LIN {X 0,Y 206.682,Z 726.89,A -85,B 0,C 180,E1 -21277.278,E2 -21277.278} C_VEL
LIN {X 0,Y 209.321,Z 735.161,A -85,B 0,C 180,E1 -21281.538,E2 -21281.538} C_VEL
LIN {X 0,Y 210.247,Z 738.551,A -85,B 0,C 180,E1 -21283.14,E2 -21283.14} C_VEL
LIN {X 0,Y 210.147,Z 740.81,A -85,B 0,C 180,E1 -21284.029,E2 -21284.029} C_VEL
LIN {X 0,Y 208.364,Z 745.04,A -85,B 0,C 180,E1 -21285.371,E2 -21285.371} C_VEL
LIN {X 0,Y 206.552,Z 749.333,A -85,B 0,C 180,E1 -21286.732,E2 -21286.732} C_VEL
LIN {X 0,Y 206.448,Z 751.668,A -85,B 0,C 180,E1 -21287.635,E2 -21287.635} C_VEL
LIN {X 0,Y 206.909,Z 753.554,A -85,B 0,C 180,E1 -21288.438,E2 -21288.438} C_VEL
LIN {X 0,Y 209.343,Z 758.765,A -85,B 0,C 180,E1 -21289.235,E2 -21289.235} C_VEL
LIN {X 0,Y 216.039,Z 774.038,A -85,B 0,C 180,E1 -21291.329,E2 -21291.329} C_VEL
LIN {X 0,Y 217.099,Z 777.167,A -85,B 0,C 180,E1 -21291.673,E2 -21291.673} C_VEL
LIN {X 0,Y 219.836,Z 802.695,A -85,B 0,C 180,E1 -21293.228,E2 -21293.228} C_VEL
LIN {X 0,Y 222.118,Z 834.204,A -85,B 0,C 180,E1 -21294.866,E2 -21294.866} C_VEL
LIN {X 0,Y 222.467,Z 842.853,A -85,B 0,C 180,E1 -21295.257,E2 -21295.257} C_VEL
LIN {X 0,Y 221.203,Z 868.34,A -85,B 0,C 180,E1 -21296.1,E2 -21296.1} C_VEL
LIN {X 0,Y 219.69,Z 881.832,A -85,B 0,C 180,E1 -21296.868,E2 -21296.868} C_VEL
LIN {X 0,Y 217.809,Z 893.498,A -85,B 0,C 180,E1 -21297.849,E2 -21297.849} C_VEL
LIN {X 0,Y 215.482,Z 904.646,A -85,B 0,C 180,E1 -21299.107,E2 -21299.107} C_VEL
LIN {X 0,Y 212.493,Z 916.272,A -85,B 0,C 180,E1 -21300.818,E2 -21300.818} C_VEL
LIN {X 0,Y 209.467,Z 926.778,A -85,B 0,C 180,E1 -21302.814,E2 -21302.814} C_VEL
LIN {X 0,Y 206.798,Z 935.404,A -85,B 0,C 180,E1 -21304.877,E2 -21304.877} C_VEL
LIN {X 0,Y 204.268,Z 943.402,A -85,B 0,C 180,E1 -21307.244,E2 -21307.244} C_VEL
LIN {X 0,Y 201.734,Z 951.707,A -85,B 0,C 180,E1 -21310.359,E2 -21310.359} C_VEL
LIN {X 0,Y 199.924,Z 958.604,A -85,B 0,C 180,E1 -21313.682,E2 -21313.682} C_VEL
LIN {X 0,Y 198.895,Z 963.537,A -85,B 0,C 180,E1 -21316.737,E2 -21316.737} C_VEL
LIN {X 0,Y 198.461,Z 967.368,A -85,B 0,C 180,E1 -21319.816,E2 -21319.816} C_VEL
LIN {X 0,Y 198.565,Z 969.739,A -85,B 0,C 180,E1 -21322.322,E2 -21322.322} C_VEL
LIN {X 0,Y 199.067,Z 972.036,A -85,B 0,C 180,E1 -21325.965,E2 -21325.965} C_VEL
LIN {X 0,Y 199.324,Z 972.723,A -85,B 0,C 180,E1 -21327.993,E2 -21327.993} C_VEL
LIN {X 0,Y 199.612,Z 972.988,A -85,B 0,C 180,E1 -21330.013,E2 -21330.013} C_VEL
LIN {X 0,Y 199.315,Z 972.703,A -85,B 0,C 180,E1 -21332.034,E2 -21332.034} C_VEL
LIN {X 0,Y 199.032,Z 971.999,A -85,B 0,C 180,E1 -21334.063,E2 -21334.063} C_VEL
LIN {X 0,Y 198.567,Z 969.697,A -85,B 0,C 180,E1 -21337.684,E2 -21337.684} C_VEL
LIN {X 0,Y 198.778,Z 965.514,A -85,B 0,C 180,E1 -21341.743,E2 -21341.743} C_VEL
LIN {X 0,Y 198.912,Z 964.926,A -85,B 0,C 180,E1 -21342.252,E2 -21342.252} C_VEL
LIN {X 0,Y 199.993,Z 963.252,A -85,B 0,C 180,E1 -21346.34,E2 -21346.34} C_VEL
LIN {X 0,Y 200.983,Z 961.887,A -85,B 0,C 180,E1 -21348.356,E2 -21348.356} C_VEL
LIN {X 0,Y 204.209,Z 958.13,A -85,B 0,C 180,E1 -21352.258,E2 -21352.258} C_VEL
LIN {X 0,Y 207.427,Z 954.488,A -85,B 0,C 180,E1 -21355.069,E2 -21355.069} C_VEL
LIN {X 0,Y 212.837,Z 948.196,A -85,B 0,C 180,E1 -21358.619,E2 -21358.619} C_VEL
LIN {X 0,Y 217.816,Z 942.411,A -85,B 0,C 180,E1 -21361.093,E2 -21361.093} C_VEL
LIN {X 0,Y 223.39,Z 935.631,A -85,B 0,C 180,E1 -21363.417,E2 -21363.417} C_VEL
LIN {X 0,Y 229.603,Z 927.592,A -85,B 0,C 180,E1 -21365.573,E2 -21365.573} C_VEL
LIN {X 0,Y 235.263,Z 919.853,A -85,B 0,C 180,E1 -21367.235,E2 -21367.235} C_VEL
LIN {X 0,Y 241.992,Z 909.858,A -85,B 0,C 180,E1 -21368.916,E2 -21368.916} C_VEL
LIN {X 0,Y 247.802,Z 900.362,A -85,B 0,C 180,E1 -21370.193,E2 -21370.193} C_VEL
LIN {X 0,Y 253.695,Z 889.722,A -85,B 0,C 180,E1 -21371.324,E2 -21371.324} C_VEL
LIN {X 0,Y 259.007,Z 879.001,A -85,B 0,C 180,E1 -21372.199,E2 -21372.199} C_VEL
LIN {X 0,Y 264.829,Z 865.221,A -85,B 0,C 180,E1 -21373.116,E2 -21373.116} C_VEL
LIN {X 0,Y 269.77,Z 850.878,A -85,B 0,C 180,E1 -21373.951,E2 -21373.951} C_VEL
LIN {X 0,Y 272.98,Z 838.674,A -85,B 0,C 180,E1 -21374.9,E2 -21374.9} C_VEL
LIN {X 0,Y 276.113,Z 825.678,A -85,B 0,C 180,E1 -21376.168,E2 -21376.168} C_VEL
LIN {X 0,Y 277.691,Z 819.801,A -85,B 0,C 180,E1 -21376.838,E2 -21376.838} C_VEL
LIN {X 0,Y 277.681,Z 819.973,A -85,B 0,C 180,E1 -21377.153,E2 -21377.153} C_VEL
LIN {X 0,Y 272.848,Z 838.879,A -85,B 0,C 180,E1 -21378.34,E2 -21378.34} C_VEL
LIN {X 0,Y 269.797,Z 848.885,A -85,B 0,C 180,E1 -21379.119,E2 -21379.119} C_VEL
LIN {X 0,Y 265.86,Z 859.286,A -85,B 0,C 180,E1 -21380.13,E2 -21380.13} C_VEL
LIN {X 0,Y 261.413,Z 869.331,A -85,B 0,C 180,E1 -21381.313,E2 -21381.313} C_VEL
LIN {X 0,Y 255.951,Z 879.698,A -85,B 0,C 180,E1 -21382.837,E2 -21382.837} C_VEL
LIN {X 0,Y 250.488,Z 888.462,A -85,B 0,C 180,E1 -21384.468,E2 -21384.468} C_VEL
LIN {X 0,Y 244.479,Z 896.754,A -85,B 0,C 180,E1 -21386.401,E2 -21386.401} C_VEL
LIN {X 0,Y 239.584,Z 902.654,A -85,B 0,C 180,E1 -21388.129,E2 -21388.129} C_VEL
LIN {X 0,Y 235.845,Z 906.785,A -85,B 0,C 180,E1 -21389.563,E2 -21389.563} C_VEL
LIN {X 0,Y 230.515,Z 911.827,A -85,B 0,C 180,E1 -21391.799,E2 -21391.799} C_VEL
LIN {X 0,Y 225.539,Z 915.826,A -85,B 0,C 180,E1 -21394.135,E2 -21394.135} C_VEL
LIN {X 0,Y 222.426,Z 917.98,A -85,B 0,C 180,E1 -21395.747,E2 -21395.747} C_VEL
LIN {X 0,Y 216.721,Z 920.844,A -85,B 0,C 180,E1 -21399.101,E2 -21399.101} C_VEL
LIN {X 0,Y 214.157,Z 921.719,A -85,B 0,C 180,E1 -21400.842,E2 -21400.842} C_VEL
LIN {X 0,Y 209.572,Z 922.218,A -85,B 0,C 180,E1 -21404.438,E2 -21404.438} C_VEL
LIN {X 0,Y 207.565,Z 921.861,A -85,B 0,C 180,E1 -21406.29,E2 -21406.29} C_VEL
LIN {X 0,Y 205.827,Z 921.101,A -85,B 0,C 180,E1 -21408.178,E2 -21408.178} C_VEL
LIN {X 0,Y 204.377,Z 919.916,A -85,B 0,C 180,E1 -21410.1,E2 -21410.1} C_VEL
LIN {X 0,Y 202.622,Z 917.373,A -85,B 0,C 180,E1 -21413.027,E2 -21413.027} C_VEL
LIN {X 0,Y 201.189,Z 913.896,A -85,B 0,C 180,E1 -21415.994,E2 -21415.994} C_VEL
LIN {X 0,Y 200.193,Z 909.353,A -85,B 0,C 180,E1 -21418.994,E2 -21418.994} C_VEL
LIN {X 0,Y 199.633,Z 903.656,A -85,B 0,C 180,E1 -21422.018,E2 -21422.018} C_VEL
LIN {X 0,Y 199.473,Z 896.674,A -85,B 0,C 180,E1 -21425.053,E2 -21425.053} C_VEL
LIN {X 0,Y 199.828,Z 889.762,A -85,B 0,C 180,E1 -21427.579,E2 -21427.579} C_VEL
LIN {X 0,Y 200.16,Z 883.329,A -85,B 0,C 180,E1 -21429.601,E2 -21429.601} C_VEL
LIN {X 0,Y 200.784,Z 873.815,A -85,B 0,C 180,E1 -21432.123,E2 -21432.123} C_VEL
LIN {X 0,Y 201.441,Z 864.862,A -85,B 0,C 180,E1 -21434.136,E2 -21434.136} C_VEL
LIN {X 0,Y 202.101,Z 855.689,A -85,B 0,C 180,E1 -21435.894,E2 -21435.894} C_VEL
LIN {X 0,Y 202.743,Z 846.48,A -85,B 0,C 180,E1 -21437.397,E2 -21437.397} C_VEL
LIN {X 0,Y 203.492,Z 835.433,A -85,B 0,C 180,E1 -21438.892,E2 -21438.892} C_VEL
LIN {X 0,Y 204.086,Z 825.218,A -85,B 0,C 180,E1 -21440.012,E2 -21440.012} C_VEL
LIN {X 0,Y 204.601,Z 813.625,A -85,B 0,C 180,E1 -21441.01,E2 -21441.01} C_VEL
LIN {X 0,Y 205.158,Z 794.728,A -85,B 0,C 180,E1 -21442.202,E2 -21442.202} C_VEL
LIN {X 0,Y 206.609,Z 752.336,A -85,B 0,C 180,E1 -21444.663,E2 -21444.663} C_VEL
LIN {X 0,Y 199.974,Z 728.514,A -85,B 0,C 180,E1 -21446.385,E2 -21446.385} C_VEL
LIN {X 0,Y 199.791,Z 727.599,A -85,B 0,C 180,E1 -21446.517,E2 -21446.517} C_VEL
LIN {X 0,Y 199.694,Z 727.61,A -85,B 0,C 180,E1 -21452.346,E2 -21452.346} C_VEL
LIN {X 0,Y 199.645,Z 727.612,A -85,B 0,C 180,E1 -21456.759,E2 -21456.759} C_VEL
LIN {X 0,Y 199.622,Z 727.614,A -85,B 0,C 180,E1 -21459.325,E2 -21459.325} C_VEL
LIN {X 0,Y 199.592,Z 727.617,A -85,B 0,C 180,E1 -21462.3,E2 -21462.3} C_VEL
LIN {X 0,Y 199.615,Z 727.614,A -85,B 0,C 180,E1 -21467.447,E2 -21467.447} C_VEL
LIN {X 0,Y 200.663,Z 730.57,A -85,B 0,C 180,E1 -21467.936,E2 -21467.936} C_VEL
LIN {X 0,Y 202.629,Z 732.841,A -85,B 0,C 180,E1 -21468.561,E2 -21468.561} C_VEL
LIN {X 0,Y 204.932,Z 736.34,A -85,B 0,C 180,E1 -21469.309,E2 -21469.309} C_VEL
LIN {X 0,Y 212.578,Z 748.515,A -85,B 0,C 180,E1 -21471.644,E2 -21471.644} C_VEL
LIN {X 0,Y 220.401,Z 762.544,A -85,B 0,C 180,E1 -21473.858,E2 -21473.858} C_VEL
LIN {X 0,Y 225.212,Z 772.505,A -85,B 0,C 180,E1 -21475.165,E2 -21475.165} C_VEL
LIN {X 0,Y 224.036,Z 814.186,A -85,B 0,C 180,E1 -21476.613,E2 -21476.613} C_VEL
LIN {X 0,Y 223.198,Z 827.888,A -85,B 0,C 180,E1 -21477.481,E2 -21477.481} C_VEL
LIN {X 0,Y 221.705,Z 840.335,A -85,B 0,C 180,E1 -21478.599,E2 -21478.599} C_VEL
LIN {X 0,Y 219.835,Z 851.709,A -85,B 0,C 180,E1 -21479.985,E2 -21479.985} C_VEL
LIN {X 0,Y 217.391,Z 863.141,A -85,B 0,C 180,E1 -21481.771,E2 -21481.771} C_VEL
LIN {X 0,Y 214.936,Z 873.23,A -85,B 0,C 180,E1 -21483.793,E2 -21483.793} C_VEL
LIN {X 0,Y 212.46,Z 882.258,A -85,B 0,C 180,E1 -21486.083,E2 -21486.083} C_VEL
LIN {X 0,Y 209.598,Z 891.036,A -85,B 0,C 180,E1 -21488.86,E2 -21488.86} C_VEL
LIN {X 0,Y 206.932,Z 898.699,A -85,B 0,C 180,E1 -21491.983,E2 -21491.983} C_VEL
LIN {X 0,Y 205.007,Z 904.459,A -85,B 0,C 180,E1 -21495.089,E2 -21495.089} C_VEL
LIN {X 0,Y 203.947,Z 907.393,A -85,B 0,C 180,E1 -21497.044,E2 -21497.044} C_VEL
LIN {X 0,Y 202.294,Z 910.949,A -85,B 0,C 180,E1 -21499.984,E2 -21499.984} C_VEL
LIN {X 0,Y 201.542,Z 912.771,A -85,B 0,C 180,E1 -21501.969,E2 -21501.969} C_VEL
LIN {X 0,Y 200.837,Z 915.075,A -85,B 0,C 180,E1 -21505.974,E2 -21505.974} C_VEL
LIN {X 0,Y 200.446,Z 915.911,A -85,B 0,C 180,E1 -21509.987,E2 -21509.987} C_VEL
LIN {X 0,Y 200.829,Z 915.143,A -85,B 0,C 180,E1 -21514,E2 -21514} C_VEL
LIN {X 0,Y 201.516,Z 912.91,A -85,B 0,C 180,E1 -21518.005,E2 -21518.005} C_VEL
LIN {X 0,Y 202.756,Z 910.086,A -85,B 0,C 180,E1 -21520.976,E2 -21520.976} C_VEL
LIN {X 0,Y 204.386,Z 906.255,A -85,B 0,C 180,E1 -21523.914,E2 -21523.914} C_VEL
LIN {X 0,Y 206.303,Z 900.776,A -85,B 0,C 180,E1 -21527.134,E2 -21527.134} C_VEL
LIN {X 0,Y 208.71,Z 893.957,A -85,B 0,C 180,E1 -21530.176,E2 -21530.176} C_VEL
LIN {X 0,Y 211.425,Z 885.922,A -85,B 0,C 180,E1 -21532.975,E2 -21532.975} C_VEL
LIN {X 0,Y 213.852,Z 877.695,A -85,B 0,C 180,E1 -21535.276,E2 -21535.276} C_VEL
LIN {X 0,Y 216.494,Z 867.509,A -85,B 0,C 180,E1 -21537.539,E2 -21537.539} C_VEL
LIN {X 0,Y 218.937,Z 857.028,A -85,B 0,C 180,E1 -21539.362,E2 -21539.362} C_VEL
LIN {X 0,Y 221.06,Z 845.742,A -85,B 0,C 180,E1 -21540.91,E2 -21540.91} C_VEL
LIN {X 0,Y 222.821,Z 833.772,A -85,B 0,C 180,E1 -21542.141,E2 -21542.141} C_VEL
LIN {X 0,Y 223.808,Z 820.26,A -85,B 0,C 180,E1 -21543.191,E2 -21543.191} C_VEL
LIN {X 0,Y 224.359,Z 807.45,A -85,B 0,C 180,E1 -21543.801,E2 -21543.801} C_VEL
LIN {X 0,Y 225.36,Z 772.626,A -85,B 0,C 180,E1 -21544.956,E2 -21544.956} C_VEL
LIN {X 0,Y 218.541,Z 759.044,A -85,B 0,C 180,E1 -21546.814,E2 -21546.814} C_VEL
LIN {X 0,Y 211.371,Z 746.467,A -85,B 0,C 180,E1 -21548.88,E2 -21548.88} C_VEL
LIN {X 0,Y 204.548,Z 735.867,A -85,B 0,C 180,E1 -21550.983,E2 -21550.983} C_VEL
LIN {X 0,Y 202.076,Z 732.119,A -85,B 0,C 180,E1 -21551.794,E2 -21551.794} C_VEL
LIN {X 0,Y 200.231,Z 729.623,A -85,B 0,C 180,E1 -21552.405,E2 -21552.405} C_VEL
LIN {X 0,Y 199.679,Z 727.604,A -85,B 0,C 180,E1 -21552.669,E2 -21552.669} C_VEL
LIN {X 0,Y 199.649,Z 727.607,A -85,B 0,C 180,E1 -21557.642,E2 -21557.642} C_VEL
LIN {X 0,Y 199.659,Z 727.607,A -85,B 0,C 180,E1 -21560.725,E2 -21560.725} C_VEL
LIN {X 0,Y 199.585,Z 727.612,A -85,B 0,C 180,E1 -21565.708,E2 -21565.708} C_VEL
LIN {X 0,Y 199.646,Z 727.616,A -85,B 0,C 180,E1 -21568.127,E2 -21568.127} C_VEL
LIN {X 0,Y 199.633,Z 727.614,A -85,B 0,C 180,E1 -21572.764,E2 -21572.764} C_VEL
LIN {X 0,Y 199.659,Z 727.602,A -85,B 0,C 180,E1 -21577.219,E2 -21577.219} C_VEL
LIN {X 0,Y 199.74,Z 727.589,A -85,B 0,C 180,E1 -21581.753,E2 -21581.753} C_VEL
LIN {X 0,Y 199.773,Z 727.602,A -85,B 0,C 180,E1 -21585.744,E2 -21585.744} C_VEL
LIN {X 0,Y 199.992,Z 727.557,A -85,B 0,C 180,E1 -21589.88,E2 -21589.88} C_VEL
LIN {X 0,Y 199.971,Z 727.576,A -85,B 0,C 180,E1 -21593.948,E2 -21593.948} C_VEL
LIN {X 0,Y 200.286,Z 727.534,A -85,B 0,C 180,E1 -21597.989,E2 -21597.989} C_VEL
LIN {X 0,Y 200.422,Z 727.525,A -85,B 0,C 180,E1 -21600,E2 -21600} C_VEL
LIN {X 0,Y 200.286,Z 727.525,A -85,B 0,C 180,E1 -21602.011,E2 -21602.011} C_VEL
LIN {X 0,Y 200.04,Z 727.557,A -85,B 0,C 180,E1 -21608.079,E2 -21608.079} C_VEL
LIN {X 0,Y 199.825,Z 727.596,A -85,B 0,C 180,E1 -21612.182,E2 -21612.182} C_VEL
LIN {X 0,Y 199.742,Z 727.601,A -85,B 0,C 180,E1 -21616.349,E2 -21616.349} C_VEL
LIN {X 0,Y 199.633,Z 727.601,A -85,B 0,C 180,E1 -21620.613,E2 -21620.613} C_VEL
LIN {X 0,Y 199.615,Z 727.609,A -85,B 0,C 180,E1 -21624.992,E2 -21624.992} C_VEL
LIN {X 0,Y 199.613,Z 727.61,A -85,B 0,C 180,E1 -21629.532,E2 -21629.532} C_VEL
LIN {X 0,Y 199.608,Z 727.621,A -85,B 0,C 180,E1 -21632.358,E2 -21632.358} C_VEL
LIN {X 0,Y 199.642,Z 727.699,A -85,B 0,C 180,E1 -21635.699,E2 -21635.699} C_VEL
LIN {X 0,Y 202.208,Z 735.817,A -85,B 0,C 180,E1 -21640.15,E2 -21640.15} C_VEL
LIN {X 0,Y 204.255,Z 743.119,A -85,B 0,C 180,E1 -21643.756,E2 -21643.756} C_VEL
LIN {X 0,Y 206.448,Z 751.668,A -85,B 0,C 180,E1 -21647.635,E2 -21647.635} C_VEL
LIN {X 0,Y 207.307,Z 754.167,A -85,B 0,C 180,E1 -21648.409,E2 -21648.409} C_VEL
LIN {X 0,Y 209.079,Z 758.994,A -85,B 0,C 180,E1 -21649.184,E2 -21649.184} C_VEL
LIN {X 0,Y 210.72,Z 766.498,A -85,B 0,C 180,E1 -21649.857,E2 -21649.857} C_VEL
LIN {X 0,Y 211.768,Z 780.813,A -85,B 0,C 180,E1 -21650.718,E2 -21650.718} C_VEL
LIN {X 0,Y 214.104,Z 803.757,A -85,B 0,C 180,E1 -21652.158,E2 -21652.158} C_VEL
LIN {X 0,Y 216.27,Z 834.897,A -85,B 0,C 180,E1 -21653.836,E2 -21653.836} C_VEL
LIN {X 0,Y 216.602,Z 842.778,A -85,B 0,C 180,E1 -21654.21,E2 -21654.21} C_VEL
LIN {X 0,Y 215.429,Z 866.419,A -85,B 0,C 180,E1 -21655.004,E2 -21655.004} C_VEL
LIN {X 0,Y 213.934,Z 879.662,A -85,B 0,C 180,E1 -21655.748,E2 -21655.748} C_VEL
LIN {X 0,Y 211.831,Z 892.491,A -85,B 0,C 180,E1 -21656.827,E2 -21656.827} C_VEL
LIN {X 0,Y 209.431,Z 903.639,A -85,B 0,C 180,E1 -21658.111,E2 -21658.111} C_VEL
LIN {X 0,Y 206.327,Z 915.264,A -85,B 0,C 180,E1 -21659.857,E2 -21659.857} C_VEL
LIN {X 0,Y 203.093,Z 925.755,A -85,B 0,C 180,E1 -21661.886,E2 -21661.886} C_VEL
LIN {X 0,Y 200.36,Z 934.389,A -85,B 0,C 180,E1 -21664.011,E2 -21664.011} C_VEL
LIN {X 0,Y 197.687,Z 942.383,A -85,B 0,C 180,E1 -21666.441,E2 -21666.441} C_VEL
LIN {X 0,Y 195.345,Z 949.874,A -85,B 0,C 180,E1 -21669.295,E2 -21669.295} C_VEL
LIN {X 0,Y 193.539,Z 955.688,A -85,B 0,C 180,E1 -21672.037,E2 -21672.037} C_VEL
LIN {X 0,Y 192.209,Z 961.006,A -85,B 0,C 180,E1 -21675.185,E2 -21675.185} C_VEL
LIN {X 0,Y 191.533,Z 965.201,A -85,B 0,C 180,E1 -21678.372,E2 -21678.372} C_VEL
LIN {X 0,Y 191.505,Z 968.884,A -85,B 0,C 180,E1 -21682.252,E2 -21682.252} C_VEL
LIN {X 0,Y 191.969,Z 971.021,A -85,B 0,C 180,E1 -21685.815,E2 -21685.815} C_VEL
LIN {X 0,Y 192.264,Z 971.716,A -85,B 0,C 180,E1 -21687.919,E2 -21687.919} C_VEL
LIN {X 0,Y 192.569,Z 971.983,A -85,B 0,C 180,E1 -21690.014,E2 -21690.014} C_VEL
LIN {X 0,Y 192.252,Z 971.695,A -85,B 0,C 180,E1 -21692.109,E2 -21692.109} C_VEL
LIN {X 0,Y 191.935,Z 970.984,A -85,B 0,C 180,E1 -21694.213,E2 -21694.213} C_VEL
LIN {X 0,Y 191.506,Z 968.843,A -85,B 0,C 180,E1 -21697.751,E2 -21697.751} C_VEL
LIN {X 0,Y 191.685,Z 965.136,A -85,B 0,C 180,E1 -21701.647,E2 -21701.647} C_VEL
LIN {X 0,Y 192.033,Z 963.462,A -85,B 0,C 180,E1 -21703.101,E2 -21703.101} C_VEL
LIN {X 0,Y 193.163,Z 962.18,A -85,B 0,C 180,E1 -21706.935,E2 -21706.935} C_VEL
LIN {X 0,Y 195.475,Z 959.665,A -85,B 0,C 180,E1 -21710.806,E2 -21710.806} C_VEL
LIN {X 0,Y 198.681,Z 956.637,A -85,B 0,C 180,E1 -21714.016,E2 -21714.016} C_VEL
LIN {X 0,Y 203.688,Z 951.595,A -85,B 0,C 180,E1 -21717.775,E2 -21717.775} C_VEL
LIN {X 0,Y 208.299,Z 946.892,A -85,B 0,C 180,E1 -21720.417,E2 -21720.417} C_VEL
LIN {X 0,Y 214.636,Z 940.191,A -85,B 0,C 180,E1 -21723.274,E2 -21723.274} C_VEL
LIN {X 0,Y 220.663,Z 933.395,A -85,B 0,C 180,E1 -21725.551,E2 -21725.551} C_VEL
LIN {X 0,Y 227.402,Z 925.323,A -85,B 0,C 180,E1 -21727.629,E2 -21727.629} C_VEL
LIN {X 0,Y 233.442,Z 917.617,A -85,B 0,C 180,E1 -21729.226,E2 -21729.226} C_VEL
LIN {X 0,Y 241.229,Z 906.64,A -85,B 0,C 180,E1 -21730.97,E2 -21730.97} C_VEL
LIN {X 0,Y 247.616,Z 896.668,A -85,B 0,C 180,E1 -21732.201,E2 -21732.201} C_VEL
LIN {X 0,Y 253.928,Z 885.682,A -85,B 0,C 180,E1 -21733.247,E2 -21733.247} C_VEL
LIN {X 0,Y 260.715,Z 872.156,A -85,B 0,C 180,E1 -21734.237,E2 -21734.237} C_VEL
LIN {X 0,Y 267.115,Z 856.327,A -85,B 0,C 180,E1 -21735.143,E2 -21735.143} C_VEL
LIN {X 0,Y 270.759,Z 845.161,A -85,B 0,C 180,E1 -21735.939,E2 -21735.939} C_VEL
LIN {X 0,Y 273.052,Z 837.373,A -85,B 0,C 180,E1 -21736.659,E2 -21736.659} C_VEL
LIN {X 0,Y 269.389,Z 849.095,A -85,B 0,C 180,E1 -21737.542,E2 -21737.542} C_VEL
LIN {X 0,Y 265.234,Z 859.664,A -85,B 0,C 180,E1 -21738.514,E2 -21738.514} C_VEL
LIN {X 0,Y 260.52,Z 869.771,A -85,B 0,C 180,E1 -21739.651,E2 -21739.651} C_VEL
LIN {X 0,Y 254.762,Z 880.196,A -85,B 0,C 180,E1 -21741.127,E2 -21741.127} C_VEL
LIN {X 0,Y 247.996,Z 890.406,A -85,B 0,C 180,E1 -21742.972,E2 -21742.972} C_VEL
LIN {X 0,Y 242.57,Z 897.51,A -85,B 0,C 180,E1 -21744.587,E2 -21744.587} C_VEL
LIN {X 0,Y 236.333,Z 904.531,A -85,B 0,C 180,E1 -21746.623,E2 -21746.623} C_VEL
LIN {X 0,Y 230.379,Z 910.327,A -85,B 0,C 180,E1 -21748.761,E2 -21748.761} C_VEL
LIN {X 0,Y 224.814,Z 914.954,A -85,B 0,C 180,E1 -21751.017,E2 -21751.017} C_VEL
LIN {X 0,Y 219.592,Z 918.523,A -85,B 0,C 180,E1 -21753.38,E2 -21753.38} C_VEL
LIN {X 0,Y 213.254,Z 921.885,A -85,B 0,C 180,E1 -21756.705,E2 -21756.705} C_VEL
LIN {X 0,Y 207.682,Z 923.485,A -85,B 0,C 180,E1 -21760.22,E2 -21760.22} C_VEL
LIN {X 0,Y 202.88,Z 923.594,A -85,B 0,C 180,E1 -21763.911,E2 -21763.911} C_VEL
LIN {X 0,Y 200.786,Z 923.028,A -85,B 0,C 180,E1 -21765.817,E2 -21765.817} C_VEL
LIN {X 0,Y 198.948,Z 922.046,A -85,B 0,C 180,E1 -21767.763,E2 -21767.763} C_VEL
LIN {X 0,Y 196.143,Z 918.897,A -85,B 0,C 180,E1 -21771.76,E2 -21771.76} C_VEL
LIN {X 0,Y 194.579,Z 915.419,A -85,B 0,C 180,E1 -21774.819,E2 -21774.819} C_VEL
LIN {X 0,Y 193.406,Z 910.946,A -85,B 0,C 180,E1 -21777.918,E2 -21777.918} C_VEL
LIN {X 0,Y 192.612,Z 904.231,A -85,B 0,C 180,E1 -21781.568,E2 -21781.568} C_VEL
LIN {X 0,Y 192.401,Z 897.087,A -85,B 0,C 180,E1 -21784.714,E2 -21784.714} C_VEL
LIN {X 0,Y 192.696,Z 890.026,A -85,B 0,C 180,E1 -21787.334,E2 -21787.334} C_VEL
LIN {X 0,Y 193.082,Z 883.516,A -85,B 0,C 180,E1 -21789.427,E2 -21789.427} C_VEL
LIN {X 0,Y 193.602,Z 874.958,A -85,B 0,C 180,E1 -21791.782,E2 -21791.782} C_VEL
LIN {X 0,Y 194.25,Z 865.987,A -85,B 0,C 180,E1 -21793.869,E2 -21793.869} C_VEL
LIN {X 0,Y 194.949,Z 856.821,A -85,B 0,C 180,E1 -21795.687,E2 -21795.687} C_VEL
LIN {X 0,Y 195.536,Z 847.567,A -85,B 0,C 180,E1 -21797.249,E2 -21797.249} C_VEL
LIN {X 0,Y 196.343,Z 836.551,A -85,B 0,C 180,E1 -21798.793,E2 -21798.793} C_VEL
LIN {X 0,Y 197.016,Z 825.184,A -85,B 0,C 180,E1 -21800.081,E2 -21800.081} C_VEL
LIN {X 0,Y 197.525,Z 813.614,A -85,B 0,C 180,E1 -21801.105,E2 -21801.105} C_VEL
LIN {X 0,Y 198.374,Z 783.132,A -85,B 0,C 180,E1 -21803.074,E2 -21803.074} C_VEL
LIN {X 0,Y 199.568,Z 753.543,A -85,B 0,C 180,E1 -21804.862,E2 -21804.862} C_VEL
LIN {X 0,Y 192.738,Z 728.477,A -85,B 0,C 180,E1 -21806.755,E2 -21806.755} C_VEL
LIN {X 0,Y 192.634,Z 728.487,A -85,B 0,C 180,E1 -21812.933,E2 -21812.933} C_VEL
LIN {X 0,Y 192.61,Z 728.488,A -85,B 0,C 180,E1 -21816.59,E2 -21816.59} C_VEL
LIN {X 0,Y 192.531,Z 728.496,A -85,B 0,C 180,E1 -21821.076,E2 -21821.076} C_VEL
LIN {X 0,Y 192.546,Z 728.505,A -85,B 0,C 180,E1 -21825.525,E2 -21825.525} C_VEL
LIN {X 0,Y 193.445,Z 731.172,A -85,B 0,C 180,E1 -21825.933,E2 -21825.933} C_VEL
LIN {X 0,Y 195.706,Z 733.846,A -85,B 0,C 180,E1 -21826.727,E2 -21826.727} C_VEL
LIN {X 0,Y 197.951,Z 737.299,A -85,B 0,C 180,E1 -21827.528,E2 -21827.528} C_VEL
LIN {X 0,Y 203.703,Z 745.873,A -85,B 0,C 180,E1 -21829.441,E2 -21829.441} C_VEL
LIN {X 0,Y 210.994,Z 758.159,A -85,B 0,C 180,E1 -21831.707,E2 -21831.707} C_VEL
LIN {X 0,Y 218.095,Z 771.897,A -85,B 0,C 180,E1 -21833.777,E2 -21833.777} C_VEL
LIN {X 0,Y 219.476,Z 774.961,A -85,B 0,C 180,E1 -21834.174,E2 -21834.174} C_VEL
LIN {X 0,Y 218.571,Z 805.347,A -85,B 0,C 180,E1 -21835.211,E2 -21835.211} C_VEL
LIN {X 0,Y 218.023,Z 819.467,A -85,B 0,C 180,E1 -21835.831,E2 -21835.831} C_VEL
LIN {X 0,Y 216.99,Z 831.806,A -85,B 0,C 180,E1 -21836.718,E2 -21836.718} C_VEL
LIN {X 0,Y 215.229,Z 844.578,A -85,B 0,C 180,E1 -21837.996,E2 -21837.996} C_VEL
LIN {X 0,Y 213.099,Z 856.132,A -85,B 0,C 180,E1 -21839.538,E2 -21839.538} C_VEL
LIN {X 0,Y 210.666,Z 866.582,A -85,B 0,C 180,E1 -21841.331,E2 -21841.331} C_VEL
LIN {X 0,Y 208.083,Z 876.168,A -85,B 0,C 180,E1 -21843.403,E2 -21843.403} C_VEL
LIN {X 0,Y 205.553,Z 884.854,A -85,B 0,C 180,E1 -21845.765,E2 -21845.765} C_VEL
LIN {X 0,Y 202.619,Z 893.348,A -85,B 0,C 180,E1 -21848.629,E2 -21848.629} C_VEL
LIN {X 0,Y 200.081,Z 900.104,A -85,B 0,C 180,E1 -21851.558,E2 -21851.558} C_VEL
LIN {X 0,Y 198.224,Z 905.463,A -85,B 0,C 180,E1 -21854.566,E2 -21854.566} C_VEL
LIN {X 0,Y 197.104,Z 908.397,A -85,B 0,C 180,E1 -21856.586,E2 -21856.586} C_VEL
LIN {X 0,Y 195.377,Z 911.953,A -85,B 0,C 180,E1 -21859.625,E2 -21859.625} C_VEL
LIN {X 0,Y 194.585,Z 913.774,A -85,B 0,C 180,E1 -21861.68,E2 -21861.68} C_VEL
LIN {X 0,Y 193.827,Z 916.078,A -85,B 0,C 180,E1 -21865.828,E2 -21865.828} C_VEL
LIN {X 0,Y 193.418,Z 916.914,A -85,B 0,C 180,E1 -21869.986,E2 -21869.986} C_VEL
LIN {X 0,Y 193.819,Z 916.145,A -85,B 0,C 180,E1 -21874.145,E2 -21874.145} C_VEL
LIN {X 0,Y 194.558,Z 913.912,A -85,B 0,C 180,E1 -21878.293,E2 -21878.293} C_VEL
LIN {X 0,Y 195.861,Z 911.088,A -85,B 0,C 180,E1 -21881.368,E2 -21881.368} C_VEL
LIN {X 0,Y 197.571,Z 907.256,A -85,B 0,C 180,E1 -21884.404,E2 -21884.404} C_VEL
LIN {X 0,Y 199.597,Z 901.777,A -85,B 0,C 180,E1 -21887.728,E2 -21887.728} C_VEL
LIN {X 0,Y 202.127,Z 894.958,A -85,B 0,C 180,E1 -21890.863,E2 -21890.863} C_VEL
LIN {X 0,Y 204.972,Z 886.922,A -85,B 0,C 180,E1 -21893.742,E2 -21893.742} C_VEL
LIN {X 0,Y 207.518,Z 878.694,A -85,B 0,C 180,E1 -21896.105,E2 -21896.105} C_VEL
LIN {X 0,Y 210.287,Z 868.507,A -85,B 0,C 180,E1 -21898.424,E2 -21898.424} C_VEL
LIN {X 0,Y 212.84,Z 858.026,A -85,B 0,C 180,E1 -21900.29,E2 -21900.29} C_VEL
LIN {X 0,Y 215.062,Z 846.738,A -85,B 0,C 180,E1 -21901.872,E2 -21901.872} C_VEL
LIN {X 0,Y 216.904,Z 834.766,A -85,B 0,C 180,E1 -21903.128,E2 -21903.128} C_VEL
LIN {X 0,Y 217.966,Z 821.212,A -85,B 0,C 180,E1 -21904.204,E2 -21904.204} C_VEL
LIN {X 0,Y 218.551,Z 808.547,A -85,B 0,C 180,E1 -21904.822,E2 -21904.822} C_VEL
LIN {X 0,Y 219.51,Z 774.785,A -85,B 0,C 180,E1 -21905.984,E2 -21905.984} C_VEL
LIN {X 0,Y 212.755,Z 761.39,A -85,B 0,C 180,E1 -21907.932,E2 -21907.932} C_VEL
LIN {X 0,Y 205.359,Z 748.49,A -85,B 0,C 180,E1 -21910.203,E2 -21910.203} C_VEL
LIN {X 0,Y 198.123,Z 737.387,A -85,B 0,C 180,E1 -21912.602,E2 -21912.602} C_VEL
LIN {X 0,Y 195.872,Z 734.06,A -85,B 0,C 180,E1 -21913.399,E2 -21913.399} C_VEL
LIN {X 0,Y 195.162,Z 733.067,A -85,B 0,C 180,E1 -21913.654,E2 -21913.654} C_VEL
LIN {X 0,Y 193.321,Z 730.758,A -85,B 0,C 180,E1 -21914.314,E2 -21914.314} C_VEL
LIN {X 0,Y 192.621,Z 728.459,A -85,B 0,C 180,E1 -21914.692,E2 -21914.692} C_VEL
LIN {X 0,Y 192.572,Z 728.495,A -85,B 0,C 180,E1 -21920.006,E2 -21920.006} C_VEL
LIN {X 0,Y 192.556,Z 728.497,A -85,B 0,C 180,E1 -21924.269,E2 -21924.269} C_VEL
LIN {X 0,Y 192.549,Z 728.495,A -85,B 0,C 180,E1 -21929.27,E2 -21929.27} C_VEL
LIN {X 0,Y 192.609,Z 728.479,A -85,B 0,C 180,E1 -21931.683,E2 -21931.683} C_VEL
LIN {X 0,Y 192.631,Z 728.475,A -85,B 0,C 180,E1 -21936.339,E2 -21936.339} C_VEL
LIN {X 0,Y 192.676,Z 728.471,A -85,B 0,C 180,E1 -21941.453,E2 -21941.453} C_VEL
LIN {X 0,Y 192.702,Z 728.481,A -85,B 0,C 180,E1 -21945.209,E2 -21945.209} C_VEL
LIN {X 0,Y 192.895,Z 728.439,A -85,B 0,C 180,E1 -21949.551,E2 -21949.551} C_VEL
LIN {X 0,Y 192.99,Z 728.445,A -85,B 0,C 180,E1 -21951.624,E2 -21951.624} C_VEL
LIN {X 0,Y 193.225,Z 728.412,A -85,B 0,C 180,E1 -21957.915,E2 -21957.915} C_VEL
LIN {X 0,Y 193.387,Z 728.401,A -85,B 0,C 180,E1 -21960,E2 -21960} C_VEL
LIN {X 0,Y 192.93,Z 728.445,A -85,B 0,C 180,E1 -21964.178,E2 -21964.178} C_VEL
LIN {X 0,Y 192.99,Z 728.433,A -85,B 0,C 180,E1 -21968.376,E2 -21968.376} C_VEL
LIN {X 0,Y 192.748,Z 728.478,A -85,B 0,C 180,E1 -21972.637,E2 -21972.637} C_VEL
LIN {X 0,Y 192.697,Z 728.478,A -85,B 0,C 180,E1 -21976.964,E2 -21976.964} C_VEL
LIN {X 0,Y 192.57,Z 728.481,A -85,B 0,C 180,E1 -21981.405,E2 -21981.405} C_VEL
LIN {X 0,Y 192.602,Z 728.49,A -85,B 0,C 180,E1 -21984.225,E2 -21984.225} C_VEL
LIN {X 0,Y 192.593,Z 728.49,A -85,B 0,C 180,E1 -21988.897,E2 -21988.897} C_VEL
LIN {X 0,Y 192.54,Z 728.587,A -85,B 0,C 180,E1 -21993.982,E2 -21993.982} C_VEL
LIN {X 0,Y 194.97,Z 736.132,A -85,B 0,C 180,E1 -21998.448,E2 -21998.448} C_VEL
LIN {X 0,Y 197.279,Z 743.979,A -85,B 0,C 180,E1 -22002.599,E2 -22002.599} C_VEL
LIN {X 0,Y 199.32,Z 752.073,A -85,B 0,C 180,E1 -22006.472,E2 -22006.472} C_VEL
LIN {X 0,Y 201.999,Z 757.443,A -85,B 0,C 180,E1 -22007.416,E2 -22007.416} C_VEL
LIN {X 0,Y 207.74,Z 770.058,A -85,B 0,C 180,E1 -22009.364,E2 -22009.364} C_VEL
LIN {X 0,Y 211.641,Z 779.541,A -85,B 0,C 180,E1 -22010.637,E2 -22010.637} C_VEL
LIN {X 0,Y 211.768,Z 780.813,A -85,B 0,C 180,E1 -22010.718,E2 -22010.718} C_VEL
LIN {X 0,Y 211.798,Z 786.652,A -85,B 0,C 180,E1 -22010.971,E2 -22010.971} C_VEL
LIN {X 0,Y 209.112,Z 806.31,A -85,B 0,C 180,E1 -22011.235,E2 -22011.235} C_VEL
LIN {X 0,Y 209.019,Z 812.183,A -85,B 0,C 180,E1 -22011.464,E2 -22011.464} C_VEL
LIN {X 0,Y 210.826,Z 842.002,A -85,B 0,C 180,E1 -22013.08,E2 -22013.08} C_VEL
LIN {X 0,Y 209.552,Z 866.277,A -85,B 0,C 180,E1 -22013.927,E2 -22013.927} C_VEL
LIN {X 0,Y 207.957,Z 879.673,A -85,B 0,C 180,E1 -22014.717,E2 -22014.717} C_VEL
LIN {X 0,Y 205.859,Z 891.474,A -85,B 0,C 180,E1 -22015.733,E2 -22015.733} C_VEL
LIN {X 0,Y 203.441,Z 902.632,A -85,B 0,C 180,E1 -22017.055,E2 -22017.055} C_VEL
LIN {X 0,Y 200.22,Z 914.255,A -85,B 0,C 180,E1 -22018.837,E2 -22018.837} C_VEL
LIN {X 0,Y 196.851,Z 924.744,A -85,B 0,C 180,E1 -22020.911,E2 -22020.911} C_VEL
LIN {X 0,Y 193.982,Z 933.376,A -85,B 0,C 180,E1 -22023.089,E2 -22023.089} C_VEL
LIN {X 0,Y 191.146,Z 941.364,A -85,B 0,C 180,E1 -22025.584,E2 -22025.584} C_VEL
LIN {X 0,Y 188.43,Z 949.498,A -85,B 0,C 180,E1 -22028.819,E2 -22028.819} C_VEL
LIN {X 0,Y 186.187,Z 956.559,A -85,B 0,C 180,E1 -22032.44,E2 -22032.44} C_VEL
LIN {X 0,Y 184.954,Z 961.492,A -85,B 0,C 180,E1 -22035.716,E2 -22035.716} C_VEL
LIN {X 0,Y 184.403,Z 965.329,A -85,B 0,C 180,E1 -22039.03,E2 -22039.03} C_VEL
LIN {X 0,Y 184.456,Z 968.012,A -85,B 0,C 180,E1 -22042.153,E2 -22042.153} C_VEL
LIN {X 0,Y 184.875,Z 970.007,A -85,B 0,C 180,E1 -22045.654,E2 -22045.654} C_VEL
LIN {X 0,Y 185.199,Z 970.707,A -85,B 0,C 180,E1 -22047.84,E2 -22047.84} C_VEL
LIN {X 0,Y 185.524,Z 970.978,A -85,B 0,C 180,E1 -22050.014,E2 -22050.014} C_VEL
LIN {X 0,Y 185.184,Z 970.686,A -85,B 0,C 180,E1 -22052.189,E2 -22052.189} C_VEL
LIN {X 0,Y 184.842,Z 969.968,A -85,B 0,C 180,E1 -22054.375,E2 -22054.375} C_VEL
LIN {X 0,Y 184.456,Z 967.972,A -85,B 0,C 180,E1 -22057.848,E2 -22057.848} C_VEL
LIN {X 0,Y 184.704,Z 964.117,A -85,B 0,C 180,E1 -22062.094,E2 -22062.094} C_VEL
LIN {X 0,Y 185.222,Z 961.977,A -85,B 0,C 180,E1 -22064.012,E2 -22064.012} C_VEL
LIN {X 0,Y 186.359,Z 961.035,A -85,B 0,C 180,E1 -22067.573,E2 -22067.573} C_VEL
LIN {X 0,Y 189.102,Z 958.752,A -85,B 0,C 180,E1 -22071.831,E2 -22071.831} C_VEL
LIN {X 0,Y 193.377,Z 955.192,A -85,B 0,C 180,E1 -22075.87,E2 -22075.87} C_VEL
LIN {X 0,Y 198.969,Z 950.263,A -85,B 0,C 180,E1 -22079.651,E2 -22079.651} C_VEL
LIN {X 0,Y 204.027,Z 945.695,A -85,B 0,C 180,E1 -22082.284,E2 -22082.284} C_VEL
LIN {X 0,Y 211.843,Z 938.118,A -85,B 0,C 180,E1 -22085.503,E2 -22085.503} C_VEL
LIN {X 0,Y 218.406,Z 931.312,A -85,B 0,C 180,E1 -22087.703,E2 -22087.703} C_VEL
LIN {X 0,Y 225.576,Z 923.288,A -85,B 0,C 180,E1 -22089.707,E2 -22089.707} C_VEL
LIN {X 0,Y 232.035,Z 915.605,A -85,B 0,C 180,E1 -22091.218,E2 -22091.218} C_VEL
LIN {X 0,Y 239.563,Z 905.61,A -85,B 0,C 180,E1 -22092.751,E2 -22092.751} C_VEL
LIN {X 0,Y 246.702,Z 895.16,A -85,B 0,C 180,E1 -22093.99,E2 -22093.99} C_VEL
LIN {X 0,Y 252.753,Z 885.191,A -85,B 0,C 180,E1 -22094.887,E2 -22094.887} C_VEL
LIN {X 0,Y 258.96,Z 873.672,A -85,B 0,C 180,E1 -22095.719,E2 -22095.719} C_VEL
LIN {X 0,Y 265.126,Z 860.14,A -85,B 0,C 180,E1 -22096.495,E2 -22096.495} C_VEL
LIN {X 0,Y 266.196,Z 857.597,A -85,B 0,C 180,E1 -22096.651,E2 -22096.651} C_VEL
LIN {X 0,Y 260.623,Z 869.34,A -85,B 0,C 180,E1 -22097.872,E2 -22097.872} C_VEL
LIN {X 0,Y 255.113,Z 879.009,A -85,B 0,C 180,E1 -22099.135,E2 -22099.135} C_VEL
LIN {X 0,Y 250.304,Z 886.365,A -85,B 0,C 180,E1 -22100.3,E2 -22100.3} C_VEL
LIN {X 0,Y 244.428,Z 894.252,A -85,B 0,C 180,E1 -22101.816,E2 -22101.816} C_VEL
LIN {X 0,Y 239.222,Z 900.378,A -85,B 0,C 180,E1 -22103.269,E2 -22103.269} C_VEL
LIN {X 0,Y 233.273,Z 906.582,A -85,B 0,C 180,E1 -22105.08,E2 -22105.08} C_VEL
LIN {X 0,Y 227.215,Z 911.991,A -85,B 0,C 180,E1 -22107.096,E2 -22107.096} C_VEL
LIN {X 0,Y 222.961,Z 915.388,A -85,B 0,C 180,E1 -22108.661,E2 -22108.661} C_VEL
LIN {X 0,Y 217.269,Z 919.179,A -85,B 0,C 180,E1 -22110.974,E2 -22110.974} C_VEL
LIN {X 0,Y 213.709,Z 921.27,A -85,B 0,C 180,E1 -22112.587,E2 -22112.587} C_VEL
LIN {X 0,Y 207.034,Z 923.984,A -85,B 0,C 180,E1 -22115.961,E2 -22115.961} C_VEL
LIN {X 0,Y 204.043,Z 924.808,A -85,B 0,C 180,E1 -22117.736,E2 -22117.736} C_VEL
LIN {X 0,Y 198.582,Z 925.227,A -85,B 0,C 180,E1 -22121.427,E2 -22121.427} C_VEL
LIN {X 0,Y 193.999,Z 924.077,A -85,B 0,C 180,E1 -22125.31,E2 -22125.31} C_VEL
LIN {X 0,Y 192.08,Z 922.913,A -85,B 0,C 180,E1 -22127.318,E2 -22127.318} C_VEL
LIN {X 0,Y 189.136,Z 919.256,A -85,B 0,C 180,E1 -22131.452,E2 -22131.452} C_VEL
LIN {X 0,Y 187.528,Z 915.487,A -85,B 0,C 180,E1 -22134.624,E2 -22134.624} C_VEL
LIN {X 0,Y 186.299,Z 910.673,A -85,B 0,C 180,E1 -22137.838,E2 -22137.838} C_VEL
LIN {X 0,Y 185.584,Z 904.706,A -85,B 0,C 180,E1 -22141.085,E2 -22141.085} C_VEL
LIN {X 0,Y 185.304,Z 898.784,A -85,B 0,C 180,E1 -22143.806,E2 -22143.806} C_VEL
LIN {X 0,Y 185.474,Z 891.789,A -85,B 0,C 180,E1 -22146.527,E2 -22146.527} C_VEL
LIN {X 0,Y 185.922,Z 885.049,A -85,B 0,C 180,E1 -22148.794,E2 -22148.794} C_VEL
LIN {X 0,Y 186.514,Z 874.904,A -85,B 0,C 180,E1 -22151.662,E2 -22151.662} C_VEL
LIN {X 0,Y 187.161,Z 865.722,A -85,B 0,C 180,E1 -22153.85,E2 -22153.85} C_VEL
LIN {X 0,Y 187.888,Z 856.436,A -85,B 0,C 180,E1 -22155.735,E2 -22155.735} C_VEL
LIN {X 0,Y 188.484,Z 846.941,A -85,B 0,C 180,E1 -22157.355,E2 -22157.355} C_VEL
LIN {X 0,Y 189.237,Z 836.615,A -85,B 0,C 180,E1 -22158.823,E2 -22158.823} C_VEL
LIN {X 0,Y 189.922,Z 825.027,A -85,B 0,C 180,E1 -22160.158,E2 -22160.158} C_VEL
LIN {X 0,Y 190.545,Z 810.515,A -85,B 0,C 180,E1 -22161.431,E2 -22161.431} C_VEL
LIN {X 0,Y 192.472,Z 754.582,A -85,B 0,C 180,E1 -22165.037,E2 -22165.037} C_VEL
LIN {X 0,Y 185.687,Z 729.354,A -85,B 0,C 180,E1 -22167.013,E2 -22167.013} C_VEL
LIN {X 0,Y 185.56,Z 729.37,A -85,B 0,C 180,E1 -22172.022,E2 -22172.022} C_VEL
LIN {X 0,Y 185.529,Z 729.372,A -85,B 0,C 180,E1 -22177.308,E2 -22177.308} C_VEL
LIN {X 0,Y 185.488,Z 729.375,A -85,B 0,C 180,E1 -22180.713,E2 -22180.713} C_VEL
LIN {X 0,Y 185.482,Z 729.374,A -85,B 0,C 180,E1 -22183.283,E2 -22183.283} C_VEL
LIN {X 0,Y 186.488,Z 732.257,A -85,B 0,C 180,E1 -22183.806,E2 -22183.806} C_VEL
LIN {X 0,Y 188.756,Z 734.658,A -85,B 0,C 180,E1 -22184.675,E2 -22184.675} C_VEL
LIN {X 0,Y 190.965,Z 738.173,A -85,B 0,C 180,E1 -22185.55,E2 -22185.55} C_VEL
LIN {X 0,Y 192.634,Z 740.549,A -85,B 0,C 180,E1 -22186.175,E2 -22186.175} C_VEL
LIN {X 0,Y 197.242,Z 747.2,A -85,B 0,C 180,E1 -22187.818,E2 -22187.818} C_VEL
LIN {X 0,Y 204.414,Z 759.004,A -85,B 0,C 180,E1 -22190.218,E2 -22190.218} C_VEL
LIN {X 0,Y 211.457,Z 772.385,A -85,B 0,C 180,E1 -22192.418,E2 -22192.418} C_VEL
LIN {X 0,Y 213.734,Z 777.117,A -85,B 0,C 180,E1 -22193.101,E2 -22193.101} C_VEL
LIN {X 0,Y 212.452,Z 815.894,A -85,B 0,C 180,E1 -22194.508,E2 -22194.508} C_VEL
LIN {X 0,Y 211.538,Z 829.317,A -85,B 0,C 180,E1 -22195.387,E2 -22195.387} C_VEL
LIN {X 0,Y 210.033,Z 841.164,A -85,B 0,C 180,E1 -22196.476,E2 -22196.476} C_VEL
LIN {X 0,Y 208.027,Z 852.581,A -85,B 0,C 180,E1 -22197.879,E2 -22197.879} C_VEL
LIN {X 0,Y 205.437,Z 863.884,A -85,B 0,C 180,E1 -22199.683,E2 -22199.683} C_VEL
LIN {X 0,Y 202.714,Z 874.197,A -85,B 0,C 180,E1 -22201.799,E2 -22201.799} C_VEL
LIN {X 0,Y 200.239,Z 882.598,A -85,B 0,C 180,E1 -22203.965,E2 -22203.965} C_VEL
LIN {X 0,Y 197.564,Z 890.35,A -85,B 0,C 180,E1 -22206.396,E2 -22206.396} C_VEL
LIN {X 0,Y 194.692,Z 898.02,A -85,B 0,C 180,E1 -22209.435,E2 -22209.435} C_VEL
LIN {X 0,Y 192.547,Z 903.648,A -85,B 0,C 180,E1 -22212.281,E2 -22212.281} C_VEL
LIN {X 0,Y 190.275,Z 909.4,A -85,B 0,C 180,E1 -22216.095,E2 -22216.095} C_VEL
LIN {X 0,Y 188.469,Z 912.956,A -85,B 0,C 180,E1 -22219.241,E2 -22219.241} C_VEL
LIN {X 0,Y 187.633,Z 914.777,A -85,B 0,C 180,E1 -22221.369,E2 -22221.369} C_VEL
LIN {X 0,Y 186.818,Z 917.081,A -85,B 0,C 180,E1 -22225.671,E2 -22225.671} C_VEL
LIN {X 0,Y 186.39,Z 917.917,A -85,B 0,C 180,E1 -22229.986,E2 -22229.986} C_VEL
LIN {X 0,Y 186.81,Z 917.147,A -85,B 0,C 180,E1 -22234.301,E2 -22234.301} C_VEL
LIN {X 0,Y 187.606,Z 914.914,A -85,B 0,C 180,E1 -22238.603,E2 -22238.603} C_VEL
LIN {X 0,Y 188.977,Z 912.089,A -85,B 0,C 180,E1 -22241.788,E2 -22241.788} C_VEL
LIN {X 0,Y 190.772,Z 908.258,A -85,B 0,C 180,E1 -22244.929,E2 -22244.929} C_VEL
LIN {X 0,Y 192.915,Z 902.778,A -85,B 0,C 180,E1 -22248.364,E2 -22248.364} C_VEL
LIN {X 0,Y 195.576,Z 895.958,A -85,B 0,C 180,E1 -22251.597,E2 -22251.597} C_VEL
LIN {X 0,Y 198.559,Z 887.922,A -85,B 0,C 180,E1 -22254.559,E2 -22254.559} C_VEL
LIN {X 0,Y 201.231,Z 879.694,A -85,B 0,C 180,E1 -22256.985,E2 -22256.985} C_VEL
LIN {X 0,Y 204.133,Z 869.506,A -85,B 0,C 180,E1 -22259.363,E2 -22259.363} C_VEL
LIN {X 0,Y 206.801,Z 859.024,A -85,B 0,C 180,E1 -22261.272,E2 -22261.272} C_VEL
LIN {X 0,Y 209.127,Z 847.735,A -85,B 0,C 180,E1 -22262.888,E2 -22262.888} C_VEL
LIN {X 0,Y 211.054,Z 835.759,A -85,B 0,C 180,E1 -22264.171,E2 -22264.171} C_VEL
LIN {X 0,Y 212.18,Z 822.251,A -85,B 0,C 180,E1 -22265.269,E2 -22265.269} C_VEL
LIN {X 0,Y 212.806,Z 809.807,A -85,B 0,C 180,E1 -22265.893,E2 -22265.893} C_VEL
LIN {X 0,Y 213.779,Z 777.081,A -85,B 0,C 180,E1 -22267.053,E2 -22267.053} C_VEL
LIN {X 0,Y 206.648,Z 762.984,A -85,B 0,C 180,E1 -22269.242,E2 -22269.242} C_VEL
LIN {X 0,Y 199.167,Z 750.183,A -85,B 0,C 180,E1 -22271.699,E2 -22271.699} C_VEL
LIN {X 0,Y 193.591,Z 741.833,A -85,B 0,C 180,E1 -22273.665,E2 -22273.665} C_VEL
LIN {X 0,Y 191.258,Z 738.344,A -85,B 0,C 180,E1 -22274.542,E2 -22274.542} C_VEL
LIN {X 0,Y 189.116,Z 735.259,A -85,B 0,C 180,E1 -22275.373,E2 -22275.373} C_VEL
LIN {X 0,Y 188.425,Z 734.208,A -85,B 0,C 180,E1 -22275.651,E2 -22275.651} C_VEL
LIN {X 0,Y 186.414,Z 731.982,A -85,B 0,C 180,E1 -22276.433,E2 -22276.433} C_VEL
LIN {X 0,Y 185.537,Z 729.351,A -85,B 0,C 180,E1 -22276.909,E2 -22276.909} C_VEL
LIN {X 0,Y 185.523,Z 729.373,A -85,B 0,C 180,E1 -22279.909,E2 -22279.909} C_VEL
LIN {X 0,Y 185.531,Z 729.372,A -85,B 0,C 180,E1 -22282.693,E2 -22282.693} C_VEL
LIN {X 0,Y 185.492,Z 729.378,A -85,B 0,C 180,E1 -22287.965,E2 -22287.965} C_VEL
LIN {X 0,Y 185.531,Z 729.359,A -85,B 0,C 180,E1 -22290.568,E2 -22290.568} C_VEL
LIN {X 0,Y 185.528,Z 729.363,A -85,B 0,C 180,E1 -22295.374,E2 -22295.374} C_VEL
LIN {X 0,Y 185.619,Z 729.352,A -85,B 0,C 180,E1 -22301.129,E2 -22301.129} C_VEL
LIN {X 0,Y 185.634,Z 729.355,A -85,B 0,C 180,E1 -22304.632,E2 -22304.632} C_VEL
LIN {X 0,Y 185.857,Z 729.316,A -85,B 0,C 180,E1 -22309.371,E2 -22309.371} C_VEL
LIN {X 0,Y 185.896,Z 729.332,A -85,B 0,C 180,E1 -22313.487,E2 -22313.487} C_VEL
LIN {X 0,Y 186.167,Z 729.29,A -85,B 0,C 180,E1 -22317.836,E2 -22317.836} C_VEL
LIN {X 0,Y 186.351,Z 729.278,A -85,B 0,C 180,E1 -22320,E2 -22320} C_VEL
LIN {X 0,Y 185.875,Z 729.325,A -85,B 0,C 180,E1 -22324.337,E2 -22324.337} C_VEL
LIN {X 0,Y 185.935,Z 729.31,A -85,B 0,C 180,E1 -22328.696,E2 -22328.696} C_VEL
LIN {X 0,Y 185.673,Z 729.356,A -85,B 0,C 180,E1 -22333.127,E2 -22333.127} C_VEL
LIN {X 0,Y 185.631,Z 729.361,A -85,B 0,C 180,E1 -22337.631,E2 -22337.631} C_VEL
LIN {X 0,Y 185.532,Z 729.363,A -85,B 0,C 180,E1 -22342.26,E2 -22342.26} C_VEL
LIN {X 0,Y 185.507,Z 729.366,A -85,B 0,C 180,E1 -22347.041,E2 -22347.041} C_VEL
LIN {X 0,Y 185.528,Z 729.365,A -85,B 0,C 180,E1 -22349.502,E2 -22349.502} C_VEL
LIN {X 0,Y 185.505,Z 729.492,A -85,B 0,C 180,E1 -22352.116,E2 -22352.116} C_VEL
LIN {X 0,Y 187.85,Z 736.794,A -85,B 0,C 180,E1 -22356.77,E2 -22356.77} C_VEL
LIN {X 0,Y 190.154,Z 744.18,A -85,B 0,C 180,E1 -22360.998,E2 -22360.998} C_VEL
LIN {X 0,Y 191.843,Z 750.676,A -85,B 0,C 180,E1 -22364.315,E2 -22364.315} C_VEL
LIN {X 0,Y 194.529,Z 756.025,A -85,B 0,C 180,E1 -22365.361,E2 -22365.361} C_VEL
LIN {X 0,Y 198.61,Z 764.351,A -85,B 0,C 180,E1 -22366.873,E2 -22366.873} C_VEL
LIN {X 0,Y 204.485,Z 777.59,A -85,B 0,C 180,E1 -22368.943,E2 -22368.943} C_VEL
LIN {X 0,Y 206.184,Z 781.876,A -85,B 0,C 180,E1 -22369.529,E2 -22369.529} C_VEL
LIN {X 0,Y 208.401,Z 804.167,A -85,B 0,C 180,E1 -22370.991,E2 -22370.991} C_VEL
LIN {X 0,Y 209.019,Z 812.183,A -85,B 0,C 180,E1 -22371.464,E2 -22371.464} C_VEL
LIN {X 0,Y 208.915,Z 818.021,A -85,B 0,C 180,E1 -22371.69,E2 -22371.69} C_VEL
LIN {X 0,Y 205.333,Z 839.535,A -85,B 0,C 180,E1 -22371.855,E2 -22371.855} C_VEL
LIN {X 0,Y 205.069,Z 843.473,A -85,B 0,C 180,E1 -22371.968,E2 -22371.968} C_VEL
LIN {X 0,Y 203.818,Z 865.272,A -85,B 0,C 180,E1 -22372.744,E2 -22372.744} C_VEL
LIN {X 0,Y 202.251,Z 878.062,A -85,B 0,C 180,E1 -22373.504,E2 -22373.504} C_VEL
LIN {X 0,Y 200.005,Z 890.463,A -85,B 0,C 180,E1 -22374.583,E2 -22374.583} C_VEL
LIN {X 0,Y 197.087,Z 903.215,A -85,B 0,C 180,E1 -22376.158,E2 -22376.158} C_VEL
LIN {X 0,Y 193.774,Z 914.548,A -85,B 0,C 180,E1 -22377.984,E2 -22377.984} C_VEL
LIN {X 0,Y 190.297,Z 924.778,A -85,B 0,C 180,E1 -22380.113,E2 -22380.113} C_VEL
LIN {X 0,Y 187.008,Z 934.056,A -85,B 0,C 180,E1 -22382.607,E2 -22382.607} C_VEL
LIN {X 0,Y 183.624,Z 943.139,A -85,B 0,C 180,E1 -22385.722,E2 -22385.722} C_VEL
LIN {X 0,Y 181.009,Z 950.446,A -85,B 0,C 180,E1 -22388.934,E2 -22388.934} C_VEL
LIN {X 0,Y 179.351,Z 955.535,A -85,B 0,C 180,E1 -22391.748,E2 -22391.748} C_VEL
LIN {X 0,Y 178.025,Z 960.471,A -85,B 0,C 180,E1 -22395.148,E2 -22395.148} C_VEL
LIN {X 0,Y 177.371,Z 964.307,A -85,B 0,C 180,E1 -22398.589,E2 -22398.589} C_VEL
LIN {X 0,Y 177.385,Z 967.174,A -85,B 0,C 180,E1 -22402.097,E2 -22402.097} C_VEL
LIN {X 0,Y 177.783,Z 968.992,A -85,B 0,C 180,E1 -22405.481,E2 -22405.481} C_VEL
LIN {X 0,Y 178.129,Z 969.698,A -85,B 0,C 180,E1 -22407.754,E2 -22407.754} C_VEL
LIN {X 0,Y 178.478,Z 969.973,A -85,B 0,C 180,E1 -22410.015,E2 -22410.015} C_VEL
LIN {X 0,Y 178.112,Z 969.676,A -85,B 0,C 180,E1 -22412.276,E2 -22412.276} C_VEL
LIN {X 0,Y 177.754,Z 968.954,A -85,B 0,C 180,E1 -22414.55,E2 -22414.55} C_VEL
LIN {X 0,Y 177.389,Z 967.128,A -85,B 0,C 180,E1 -22417.911,E2 -22417.911} C_VEL
LIN {X 0,Y 177.525,Z 964.24,A -85,B 0,C 180,E1 -22421.431,E2 -22421.431} C_VEL
LIN {X 0,Y 178.501,Z 960.379,A -85,B 0,C 180,E1 -22424.988,E2 -22424.988} C_VEL
LIN {X 0,Y 179.588,Z 959.786,A -85,B 0,C 180,E1 -22428.259,E2 -22428.259} C_VEL
LIN {X 0,Y 182.539,Z 957.864,A -85,B 0,C 180,E1 -22432.659,E2 -22432.659} C_VEL
LIN {X 0,Y 187.011,Z 954.654,A -85,B 0,C 180,E1 -22436.82,E2 -22436.82} C_VEL
LIN {X 0,Y 191.252,Z 951.462,A -85,B 0,C 180,E1 -22439.755,E2 -22439.755} C_VEL
LIN {X 0,Y 196.213,Z 947.539,A -85,B 0,C 180,E1 -22442.512,E2 -22442.512} C_VEL
LIN {X 0,Y 201.994,Z 942.828,A -85,B 0,C 180,E1 -22445.049,E2 -22445.049} C_VEL
LIN {X 0,Y 209.412,Z 936.199,A -85,B 0,C 180,E1 -22447.782,E2 -22447.782} C_VEL
LIN {X 0,Y 217.743,Z 928.161,A -85,B 0,C 180,E1 -22450.218,E2 -22450.218} C_VEL
LIN {X 0,Y 224.165,Z 921.483,A -85,B 0,C 180,E1 -22451.789,E2 -22451.789} C_VEL
LIN {X 0,Y 231.924,Z 912.696,A -85,B 0,C 180,E1 -22453.4,E2 -22453.4} C_VEL
LIN {X 0,Y 239.532,Z 903.051,A -85,B 0,C 180,E1 -22454.775,E2 -22454.775} C_VEL
LIN {X 0,Y 246.314,Z 893.649,A -85,B 0,C 180,E1 -22455.809,E2 -22455.809} C_VEL
LIN {X 0,Y 252.641,Z 883.739,A -85,B 0,C 180,E1 -22456.626,E2 -22456.626} C_VEL
LIN {X 0,Y 255.028,Z 879.756,A -85,B 0,C 180,E1 -22456.921,E2 -22456.921} C_VEL
LIN {X 0,Y 255.417,Z 878.953,A -85,B 0,C 180,E1 -22457.308,E2 -22457.308} C_VEL
LIN {X 0,Y 249.606,Z 887.427,A -85,B 0,C 180,E1 -22458.572,E2 -22458.572} C_VEL
LIN {X 0,Y 243.448,Z 895.3,A -85,B 0,C 180,E1 -22460.034,E2 -22460.034} C_VEL
LIN {X 0,Y 237.404,Z 901.987,A -85,B 0,C 180,E1 -22461.561,E2 -22461.561} C_VEL
LIN {X 0,Y 231.599,Z 907.706,A -85,B 0,C 180,E1 -22463.178,E2 -22463.178} C_VEL
LIN {X 0,Y 225.978,Z 912.527,A -85,B 0,C 180,E1 -22464.875,E2 -22464.875} C_VEL
LIN {X 0,Y 219.553,Z 917.271,A -85,B 0,C 180,E1 -22467.031,E2 -22467.031} C_VEL
LIN {X 0,Y 215.477,Z 919.934,A -85,B 0,C 180,E1 -22468.543,E2 -22468.543} C_VEL
LIN {X 0,Y 207.792,Z 923.749,A -85,B 0,C 180,E1 -22471.737,E2 -22471.737} C_VEL
LIN {X 0,Y 204.247,Z 925.159,A -85,B 0,C 180,E1 -22473.428,E2 -22473.428} C_VEL
LIN {X 0,Y 197.712,Z 926.6,A -85,B 0,C 180,E1 -22476.982,E2 -22476.982} C_VEL
LIN {X 0,Y 192.008,Z 926.619,A -85,B 0,C 180,E1 -22480.766,E2 -22480.766} C_VEL
LIN {X 0,Y 187.211,Z 925.008,A -85,B 0,C 180,E1 -22484.765,E2 -22484.765} C_VEL
LIN {X 0,Y 183.569,Z 921.836,A -85,B 0,C 180,E1 -22488.964,E2 -22488.964} C_VEL
LIN {X 0,Y 181.026,Z 916.948,A -85,B 0,C 180,E1 -22493.312,E2 -22493.312} C_VEL
LIN {X 0,Y 179.604,Z 912.161,A -85,B 0,C 180,E1 -22496.635,E2 -22496.635} C_VEL
LIN {X 0,Y 178.734,Z 907.363,A -85,B 0,C 180,E1 -22499.437,E2 -22499.437} C_VEL
LIN {X 0,Y 178.276,Z 900.346,A -85,B 0,C 180,E1 -22502.825,E2 -22502.825} C_VEL
LIN {X 0,Y 178.303,Z 893.443,A -85,B 0,C 180,E1 -22505.655,E2 -22505.655} C_VEL
LIN {X 0,Y 178.824,Z 885.392,A -85,B 0,C 180,E1 -22508.475,E2 -22508.475} C_VEL
LIN {X 0,Y 179.232,Z 877.305,A -85,B 0,C 180,E1 -22510.865,E2 -22510.865} C_VEL
LIN {X 0,Y 179.903,Z 867.765,A -85,B 0,C 180,E1 -22513.268,E2 -22513.268} C_VEL
LIN {X 0,Y 180.7,Z 857.168,A -85,B 0,C 180,E1 -22515.509,E2 -22515.509} C_VEL
LIN {X 0,Y 181.456,Z 845.998,A -85,B 0,C 180,E1 -22517.468,E2 -22517.468} C_VEL
LIN {X 0,Y 182.413,Z 832.258,A -85,B 0,C 180,E1 -22519.409,E2 -22519.409} C_VEL
LIN {X 0,Y 183.12,Z 818.225,A -85,B 0,C 180,E1 -22520.868,E2 -22520.868} C_VEL
LIN {X 0,Y 183.694,Z 802.6,A -85,B 0,C 180,E1 -22522.05,E2 -22522.05} C_VEL
LIN {X 0,Y 185.307,Z 755.3,A -85,B 0,C 180,E1 -22525.224,E2 -22525.224} C_VEL
LIN {X 0,Y 178.62,Z 730.233,A -85,B 0,C 180,E1 -22527.264,E2 -22527.264} C_VEL
LIN {X 0,Y 178.513,Z 730.244,A -85,B 0,C 180,E1 -22533.448,E2 -22533.448} C_VEL
LIN {X 0,Y 178.415,Z 730.254,A -85,B 0,C 180,E1 -22539.07,E2 -22539.07} C_VEL
LIN {X 0,Y 178.461,Z 730.354,A -85,B 0,C 180,E1 -22540.826,E2 -22540.826} C_VEL
LIN {X 0,Y 179.366,Z 733.024,A -85,B 0,C 180,E1 -22541.333,E2 -22541.333} C_VEL
LIN {X 0,Y 181.469,Z 735.23,A -85,B 0,C 180,E1 -22542.24,E2 -22542.24} C_VEL
LIN {X 0,Y 182.551,Z 737.027,A -85,B 0,C 180,E1 -22542.73,E2 -22542.73} C_VEL
LIN {X 0,Y 185.472,Z 740.854,A -85,B 0,C 180,E1 -22543.947,E2 -22543.947} C_VEL
LIN {X 0,Y 192.974,Z 751.852,A -85,B 0,C 180,E1 -22546.853,E2 -22546.853} C_VEL
LIN {X 0,Y 200.189,Z 763.943,A -85,B 0,C 180,E1 -22549.398,E2 -22549.398} C_VEL
LIN {X 0,Y 207.04,Z 777.288,A -85,B 0,C 180,E1 -22551.65,E2 -22551.65} C_VEL
LIN {X 0,Y 208.058,Z 779.441,A -85,B 0,C 180,E1 -22551.974,E2 -22551.974} C_VEL
LIN {X 0,Y 206.7,Z 817.863,A -85,B 0,C 180,E1 -22553.426,E2 -22553.426} C_VEL
LIN {X 0,Y 205.712,Z 831.141,A -85,B 0,C 180,E1 -22554.341,E2 -22554.341} C_VEL
LIN {X 0,Y 204,Z 843.364,A -85,B 0,C 180,E1 -22555.511,E2 -22555.511} C_VEL
LIN {X 0,Y 201.855,Z 854.733,A -85,B 0,C 180,E1 -22556.99,E2 -22556.99} C_VEL
LIN {X 0,Y 199.065,Z 866.162,A -85,B 0,C 180,E1 -22558.9,E2 -22558.9} C_VEL
LIN {X 0,Y 196.241,Z 876.248,A -85,B 0,C 180,E1 -22561.074,E2 -22561.074} C_VEL
LIN {X 0,Y 193.376,Z 885.274,A -85,B 0,C 180,E1 -22563.55,E2 -22563.55} C_VEL
LIN {X 0,Y 190.086,Z 894.05,A -85,B 0,C 180,E1 -22566.567,E2 -22566.567} C_VEL
LIN {X 0,Y 186.996,Z 901.712,A -85,B 0,C 180,E1 -22569.984,E2 -22569.984} C_VEL
LIN {X 0,Y 184.712,Z 907.471,A -85,B 0,C 180,E1 -22573.406,E2 -22573.406} C_VEL
LIN {X 0,Y 183.46,Z 910.404,A -85,B 0,C 180,E1 -22575.568,E2 -22575.568} C_VEL
LIN {X 0,Y 181.569,Z 913.96,A -85,B 0,C 180,E1 -22578.827,E2 -22578.827} C_VEL
LIN {X 0,Y 180.687,Z 915.781,A -85,B 0,C 180,E1 -22581.035,E2 -22581.035} C_VEL
LIN {X 0,Y 179.811,Z 918.084,A -85,B 0,C 180,E1 -22585.502,E2 -22585.502} C_VEL
LIN {X 0,Y 179.363,Z 918.919,A -85,B 0,C 180,E1 -22589.985,E2 -22589.985} C_VEL
LIN {X 0,Y 179.802,Z 918.15,A -85,B 0,C 180,E1 -22594.468,E2 -22594.468} C_VEL
LIN {X 0,Y 180.659,Z 915.916,A -85,B 0,C 180,E1 -22598.936,E2 -22598.936} C_VEL
LIN {X 0,Y 182.103,Z 913.091,A -85,B 0,C 180,E1 -22602.239,E2 -22602.239} C_VEL
LIN {X 0,Y 183.99,Z 909.259,A -85,B 0,C 180,E1 -22605.492,E2 -22605.492} C_VEL
LIN {X 0,Y 186.258,Z 903.779,A -85,B 0,C 180,E1 -22609.045,E2 -22609.045} C_VEL
LIN {X 0,Y 189.059,Z 896.959,A -85,B 0,C 180,E1 -22612.38,E2 -22612.38} C_VEL
LIN {X 0,Y 192.189,Z 888.922,A -85,B 0,C 180,E1 -22615.43,E2 -22615.43} C_VEL
LIN {X 0,Y 194.995,Z 880.694,A -85,B 0,C 180,E1 -22617.922,E2 -22617.922} C_VEL
LIN {X 0,Y 198.037,Z 870.505,A -85,B 0,C 180,E1 -22620.36,E2 -22620.36} C_VEL
LIN {X 0,Y 200.826,Z 860.022,A -85,B 0,C 180,E1 -22622.313,E2 -22622.313} C_VEL
LIN {X 0,Y 203.261,Z 848.732,A -85,B 0,C 180,E1 -22623.964,E2 -22623.964} C_VEL
LIN {X 0,Y 205.278,Z 836.753,A -85,B 0,C 180,E1 -22625.273,E2 -22625.273} C_VEL
LIN {X 0,Y 206.469,Z 823.536,A -85,B 0,C 180,E1 -22626.373,E2 -22626.373} C_VEL
LIN {X 0,Y 207.135,Z 811.037,A -85,B 0,C 180,E1 -22627.024,E2 -22627.024} C_VEL
LIN {X 0,Y 208.212,Z 779.573,A -85,B 0,C 180,E1 -22628.153,E2 -22628.153} C_VEL
LIN {X 0,Y 201.178,Z 765.761,A -85,B 0,C 180,E1 -22630.443,E2 -22630.443} C_VEL
LIN {X 0,Y 194.913,Z 754.941,A -85,B 0,C 180,E1 -22632.626,E2 -22632.626} C_VEL
LIN {X 0,Y 189.269,Z 746.353,A -85,B 0,C 180,E1 -22634.731,E2 -22634.731} C_VEL
LIN {X 0,Y 187.02,Z 743.096,A -85,B 0,C 180,E1 -22635.62,E2 -22635.62} C_VEL
LIN {X 0,Y 184.424,Z 739.381,A -85,B 0,C 180,E1 -22636.69,E2 -22636.69} C_VEL
LIN {X 0,Y 182.215,Z 736.235,A -85,B 0,C 180,E1 -22637.641,E2 -22637.641} C_VEL
LIN {X 0,Y 181.579,Z 735.263,A -85,B 0,C 180,E1 -22637.927,E2 -22637.927} C_VEL
LIN {X 0,Y 179.526,Z 733.128,A -85,B 0,C 180,E1 -22638.813,E2 -22638.813} C_VEL
LIN {X 0,Y 178.557,Z 730.644,A -85,B 0,C 180,E1 -22639.336,E2 -22639.336} C_VEL
LIN {X 0,Y 178.509,Z 730.251,A -85,B 0,C 180,E1 -22639.487,E2 -22639.487} C_VEL
LIN {X 0,Y 178.443,Z 730.258,A -85,B 0,C 180,E1 -22643.787,E2 -22643.787} C_VEL
LIN {X 0,Y 178.442,Z 730.246,A -85,B 0,C 180,E1 -22646.537,E2 -22646.537} C_VEL
LIN {X 0,Y 178.472,Z 730.241,A -85,B 0,C 180,E1 -22649.998,E2 -22649.998} C_VEL
LIN {X 0,Y 178.468,Z 730.247,A -85,B 0,C 180,E1 -22654.878,E2 -22654.878} C_VEL
LIN {X 0,Y 178.567,Z 730.234,A -85,B 0,C 180,E1 -22660.78,E2 -22660.78} C_VEL
LIN {X 0,Y 178.599,Z 730.241,A -85,B 0,C 180,E1 -22666.343,E2 -22666.343} C_VEL
LIN {X 0,Y 178.867,Z 730.195,A -85,B 0,C 180,E1 -22670.957,E2 -22670.957} C_VEL
LIN {X 0,Y 179.111,Z 730.167,A -85,B 0,C 180,E1 -22677.751,E2 -22677.751} C_VEL
LIN {X 0,Y 179.315,Z 730.155,A -85,B 0,C 180,E1 -22680,E2 -22680} C_VEL
LIN {X 0,Y 178.822,Z 730.205,A -85,B 0,C 180,E1 -22684.508,E2 -22684.508} C_VEL
LIN {X 0,Y 178.867,Z 730.189,A -85,B 0,C 180,E1 -22689.042,E2 -22689.042} C_VEL
LIN {X 0,Y 178.6,Z 730.236,A -85,B 0,C 180,E1 -22693.657,E2 -22693.657} C_VEL
LIN {X 0,Y 178.566,Z 730.233,A -85,B 0,C 180,E1 -22699.22,E2 -22699.22} C_VEL
LIN {X 0,Y 178.468,Z 730.241,A -85,B 0,C 180,E1 -22705.122,E2 -22705.122} C_VEL
LIN {X 0,Y 178.478,Z 730.347,A -85,B 0,C 180,E1 -22710.005,E2 -22710.005} C_VEL
LIN {X 0,Y 181.125,Z 738.442,A -85,B 0,C 180,E1 -22715.593,E2 -22715.593} C_VEL
LIN {X 0,Y 183.639,Z 746.787,A -85,B 0,C 180,E1 -22720.587,E2 -22720.587} C_VEL
LIN {X 0,Y 184.297,Z 749.235,A -85,B 0,C 180,E1 -22721.863,E2 -22721.863} C_VEL
LIN {X 0,Y 187.008,Z 754.432,A -85,B 0,C 180,E1 -22723.033,E2 -22723.033} C_VEL
LIN {X 0,Y 191.45,Z 763.138,A -85,B 0,C 180,E1 -22724.84,E2 -22724.84} C_VEL
LIN {X 0,Y 195.822,Z 772.381,A -85,B 0,C 180,E1 -22726.523,E2 -22726.523} C_VEL
LIN {X 0,Y 200.896,Z 784.48,A -85,B 0,C 180,E1 -22728.395,E2 -22728.395} C_VEL
LIN {X 0,Y 202.983,Z 807.395,A -85,B 0,C 180,E1 -22729.929,E2 -22729.929} C_VEL
LIN {X 0,Y 204.836,Z 837.458,A -85,B 0,C 180,E1 -22731.659,E2 -22731.659} C_VEL
LIN {X 0,Y 205.069,Z 843.473,A -85,B 0,C 180,E1 -22731.968,E2 -22731.968} C_VEL
LIN {X 0,Y 204.384,Z 849.322,A -85,B 0,C 180,E1 -22732.068,E2 -22732.068} C_VEL
LIN {X 0,Y 201.64,Z 858.833,A -85,B 0,C 180,E1 -22731.915,E2 -22731.915} C_VEL
LIN {X 0,Y 198.458,Z 868.251,A -85,B 0,C 180,E1 -22731.834,E2 -22731.834} C_VEL
LIN {X 0,Y 197.088,Z 873.961,A -85,B 0,C 180,E1 -22732.058,E2 -22732.058} C_VEL
LIN {X 0,Y 194.718,Z 887.214,A -85,B 0,C 180,E1 -22733.147,E2 -22733.147} C_VEL
LIN {X 0,Y 192.087,Z 898.935,A -85,B 0,C 180,E1 -22734.511,E2 -22734.511} C_VEL
LIN {X 0,Y 188.557,Z 910.923,A -85,B 0,C 180,E1 -22736.348,E2 -22736.348} C_VEL
LIN {X 0,Y 184.987,Z 921.649,A -85,B 0,C 180,E1 -22738.527,E2 -22738.527} C_VEL
LIN {X 0,Y 181.376,Z 931.346,A -85,B 0,C 180,E1 -22741.049,E2 -22741.049} C_VEL
LIN {X 0,Y 178.219,Z 939.328,A -85,B 0,C 180,E1 -22743.682,E2 -22743.682} C_VEL
LIN {X 0,Y 175.162,Z 947.363,A -85,B 0,C 180,E1 -22747.078,E2 -22747.078} C_VEL
LIN {X 0,Y 172.547,Z 954.512,A -85,B 0,C 180,E1 -22751.001,E2 -22751.001} C_VEL
LIN {X 0,Y 171.1,Z 959.449,A -85,B 0,C 180,E1 -22754.532,E2 -22754.532} C_VEL
LIN {X 0,Y 170.363,Z 963.287,A -85,B 0,C 180,E1 -22758.113,E2 -22758.113} C_VEL
LIN {X 0,Y 170.332,Z 966.31,A -85,B 0,C 180,E1 -22761.995,E2 -22761.995} C_VEL
LIN {X 0,Y 170.696,Z 967.978,A -85,B 0,C 180,E1 -22765.293,E2 -22765.293} C_VEL
LIN {X 0,Y 171.056,Z 968.688,A -85,B 0,C 180,E1 -22767.661,E2 -22767.661} C_VEL
LIN {X 0,Y 171.429,Z 968.967,A -85,B 0,C 180,E1 -22770.016,E2 -22770.016} C_VEL
LIN {X 0,Y 171.036,Z 968.665,A -85,B 0,C 180,E1 -22772.37,E2 -22772.37} C_VEL
LIN {X 0,Y 170.67,Z 967.94,A -85,B 0,C 180,E1 -22774.739,E2 -22774.739} C_VEL
LIN {X 0,Y 170.333,Z 966.267,A -85,B 0,C 180,E1 -22778.007,E2 -22778.007} C_VEL
LIN {X 0,Y 170.526,Z 963.22,A -85,B 0,C 180,E1 -22781.907,E2 -22781.907} C_VEL
LIN {X 0,Y 171.825,Z 958.703,A -85,B 0,C 180,E1 -22786.042,E2 -22786.042} C_VEL
LIN {X 0,Y 172.872,Z 958.394,A -85,B 0,C 180,E1 -22788.995,E2 -22788.995} C_VEL
LIN {X 0,Y 176.017,Z 956.86,A -85,B 0,C 180,E1 -22793.548,E2 -22793.548} C_VEL
LIN {X 0,Y 180.706,Z 954.092,A -85,B 0,C 180,E1 -22797.835,E2 -22797.835} C_VEL
LIN {X 0,Y 185.126,Z 951.306,A -85,B 0,C 180,E1 -22800.845,E2 -22800.845} C_VEL
LIN {X 0,Y 192.2,Z 946.375,A -85,B 0,C 180,E1 -22804.54,E2 -22804.54} C_VEL
LIN {X 0,Y 200.541,Z 940.087,A -85,B 0,C 180,E1 -22807.842,E2 -22807.842} C_VEL
LIN {X 0,Y 207.459,Z 934.414,A -85,B 0,C 180,E1 -22810.078,E2 -22810.078} C_VEL
LIN {X 0,Y 216.32,Z 926.457,A -85,B 0,C 180,E1 -22812.401,E2 -22812.401} C_VEL
LIN {X 0,Y 223.131,Z 919.883,A -85,B 0,C 180,E1 -22813.876,E2 -22813.876} C_VEL
LIN {X 0,Y 232.589,Z 909.666,A -85,B 0,C 180,E1 -22815.614,E2 -22815.614} C_VEL
LIN {X 0,Y 239.225,Z 901.711,A -85,B 0,C 180,E1 -22816.657,E2 -22816.657} C_VEL
LIN {X 0,Y 244.85,Z 894.473,A -85,B 0,C 180,E1 -22817.424,E2 -22817.424} C_VEL
LIN {X 0,Y 244.188,Z 895.051,A -85,B 0,C 180,E1 -22817.961,E2 -22817.961} C_VEL
LIN {X 0,Y 236.434,Z 903.274,A -85,B 0,C 180,E1 -22819.72,E2 -22819.72} C_VEL
LIN {X 0,Y 230.278,Z 908.979,A -85,B 0,C 180,E1 -22821.27,E2 -22821.27} C_VEL
LIN {X 0,Y 223.15,Z 914.685,A -85,B 0,C 180,E1 -22823.245,E2 -22823.245} C_VEL
LIN {X 0,Y 216.334,Z 919.26,A -85,B 0,C 180,E1 -22825.353,E2 -22825.353} C_VEL
LIN {X 0,Y 209.914,Z 922.865,A -85,B 0,C 180,E1 -22827.609,E2 -22827.609} C_VEL
LIN {X 0,Y 205.85,Z 924.799,A -85,B 0,C 180,E1 -22829.195,E2 -22829.195} C_VEL
LIN {X 0,Y 198.199,Z 927.293,A -85,B 0,C 180,E1 -22832.55,E2 -22832.55} C_VEL
LIN {X 0,Y 194.699,Z 928.048,A -85,B 0,C 180,E1 -22834.332,E2 -22834.332} C_VEL
LIN {X 0,Y 188.301,Z 928.298,A -85,B 0,C 180,E1 -22838.085,E2 -22838.085} C_VEL
LIN {X 0,Y 182.829,Z 927.037,A -85,B 0,C 180,E1 -22842.09,E2 -22842.09} C_VEL
LIN {X 0,Y 180.439,Z 925.835,A -85,B 0,C 180,E1 -22844.178,E2 -22844.178} C_VEL
LIN {X 0,Y 176.612,Z 922.146,A -85,B 0,C 180,E1 -22848.523,E2 -22848.523} C_VEL
LIN {X 0,Y 174.526,Z 918.364,A -85,B 0,C 180,E1 -22851.898,E2 -22851.898} C_VEL
LIN {X 0,Y 172.867,Z 913.592,A -85,B 0,C 180,E1 -22855.336,E2 -22855.336} C_VEL
LIN {X 0,Y 171.807,Z 907.687,A -85,B 0,C 180,E1 -22858.828,E2 -22858.828} C_VEL
LIN {X 0,Y 171.32,Z 901.866,A -85,B 0,C 180,E1 -22861.763,E2 -22861.763} C_VEL
LIN {X 0,Y 171.212,Z 895.021,A -85,B 0,C 180,E1 -22864.709,E2 -22864.709} C_VEL
LIN {X 0,Y 171.625,Z 886.995,A -85,B 0,C 180,E1 -22867.648,E2 -22867.648} C_VEL
LIN {X 0,Y 172.068,Z 878.268,A -85,B 0,C 180,E1 -22870.362,E2 -22870.362} C_VEL
LIN {X 0,Y 172.755,Z 868.547,A -85,B 0,C 180,E1 -22872.928,E2 -22872.928} C_VEL
LIN {X 0,Y 173.435,Z 859.341,A -85,B 0,C 180,E1 -22874.971,E2 -22874.971} C_VEL
LIN {X 0,Y 174.033,Z 850.053,A -85,B 0,C 180,E1 -22876.722,E2 -22876.722} C_VEL
LIN {X 0,Y 174.964,Z 838.063,A -85,B 0,C 180,E1 -22878.593,E2 -22878.593} C_VEL
LIN {X 0,Y 175.764,Z 823.98,A -85,B 0,C 180,E1 -22880.327,E2 -22880.327} C_VEL
LIN {X 0,Y 176.459,Z 808.212,A -85,B 0,C 180,E1 -22881.694,E2 -22881.694} C_VEL
LIN {X 0,Y 178.254,Z 756.385,A -85,B 0,C 180,E1 -22885.402,E2 -22885.402} C_VEL
LIN {X 0,Y 171.574,Z 731.135,A -85,B 0,C 180,E1 -22887.47,E2 -22887.47} C_VEL
LIN {X 0,Y 171.439,Z 731.13,A -85,B 0,C 180,E1 -22892.204,E2 -22892.204} C_VEL
LIN {X 0,Y 171.389,Z 731.133,A -85,B 0,C 180,E1 -22897.218,E2 -22897.218} C_VEL
LIN {X 0,Y 171.396,Z 731.193,A -85,B 0,C 180,E1 -22897.957,E2 -22897.957} C_VEL
LIN {X 0,Y 172.264,Z 733.743,A -85,B 0,C 180,E1 -22898.511,E2 -22898.511} C_VEL
LIN {X 0,Y 174.18,Z 735.955,A -85,B 0,C 180,E1 -22899.469,E2 -22899.469} C_VEL
LIN {X 0,Y 175.079,Z 736.725,A -85,B 0,C 180,E1 -22899.888,E2 -22899.888} C_VEL
LIN {X 0,Y 177.112,Z 740.024,A -85,B 0,C 180,E1 -22900.902,E2 -22900.902} C_VEL
LIN {X 0,Y 178.614,Z 741.721,A -85,B 0,C 180,E1 -22901.578,E2 -22901.578} C_VEL
LIN {X 0,Y 182.481,Z 747.292,A -85,B 0,C 180,E1 -22903.297,E2 -22903.297} C_VEL
LIN {X 0,Y 188.979,Z 756.89,A -85,B 0,C 180,E1 -22905.93,E2 -22905.93} C_VEL
LIN {X 0,Y 196.057,Z 768.949,A -85,B 0,C 180,E1 -22908.559,E2 -22908.559} C_VEL
LIN {X 0,Y 202.495,Z 781.822,A -85,B 0,C 180,E1 -22910.794,E2 -22910.794} C_VEL
LIN {X 0,Y 201.131,Z 818.232,A -85,B 0,C 180,E1 -22912.194,E2 -22912.194} C_VEL
LIN {X 0,Y 200.099,Z 831.572,A -85,B 0,C 180,E1 -22913.118,E2 -22913.118} C_VEL
LIN {X 0,Y 198.251,Z 844.373,A -85,B 0,C 180,E1 -22914.362,E2 -22914.362} C_VEL
LIN {X 0,Y 195.999,Z 855.741,A -85,B 0,C 180,E1 -22915.871,E2 -22915.871} C_VEL
LIN {X 0,Y 193.081,Z 867.169,A -85,B 0,C 180,E1 -22917.823,E2 -22917.823} C_VEL
LIN {X 0,Y 190.12,Z 877.254,A -85,B 0,C 180,E1 -22920.049,E2 -22920.049} C_VEL
LIN {X 0,Y 187.11,Z 886.279,A -85,B 0,C 180,E1 -22922.591,E2 -22922.591} C_VEL
LIN {X 0,Y 183.659,Z 895.055,A -85,B 0,C 180,E1 -22925.695,E2 -22925.695} C_VEL
LIN {X 0,Y 180.409,Z 902.716,A -85,B 0,C 180,E1 -22929.22,E2 -22929.22} C_VEL
LIN {X 0,Y 177.988,Z 908.475,A -85,B 0,C 180,E1 -22932.759,E2 -22932.759} C_VEL
LIN {X 0,Y 176.663,Z 911.408,A -85,B 0,C 180,E1 -22934.999,E2 -22934.999} C_VEL
LIN {X 0,Y 174.68,Z 914.963,A -85,B 0,C 180,E1 -22938.38,E2 -22938.38} C_VEL
LIN {X 0,Y 173.748,Z 916.784,A -85,B 0,C 180,E1 -22940.674,E2 -22940.674} C_VEL
LIN {X 0,Y 172.805,Z 919.087,A -85,B 0,C 180,E1 -22945.319,E2 -22945.319} C_VEL
LIN {X 0,Y 172.335,Z 919.922,A -85,B 0,C 180,E1 -22949.985,E2 -22949.985} C_VEL
LIN {X 0,Y 172.797,Z 919.152,A -85,B 0,C 180,E1 -22954.65,E2 -22954.65} C_VEL
LIN {X 0,Y 173.72,Z 916.918,A -85,B 0,C 180,E1 -22959.297,E2 -22959.297} C_VEL
LIN {X 0,Y 175.241,Z 914.093,A -85,B 0,C 180,E1 -22962.726,E2 -22962.726} C_VEL
LIN {X 0,Y 177.227,Z 910.261,A -85,B 0,C 180,E1 -22966.099,E2 -22966.099} C_VEL
LIN {X 0,Y 179.629,Z 904.78,A -85,B 0,C 180,E1 -22969.777,E2 -22969.777} C_VEL
LIN {X 0,Y 182.58,Z 897.96,A -85,B 0,C 180,E1 -22973.22,E2 -22973.22} C_VEL
LIN {X 0,Y 185.866,Z 889.922,A -85,B 0,C 180,E1 -22976.36,E2 -22976.36} C_VEL
LIN {X 0,Y 188.815,Z 881.693,A -85,B 0,C 180,E1 -22978.921,E2 -22978.921} C_VEL
LIN {X 0,Y 192.006,Z 871.504,A -85,B 0,C 180,E1 -22981.421,E2 -22981.421} C_VEL
LIN {X 0,Y 194.922,Z 861.02,A -85,B 0,C 180,E1 -22983.417,E2 -22983.417} C_VEL
LIN {X 0,Y 197.471,Z 849.728,A -85,B 0,C 180,E1 -22985.103,E2 -22985.103} C_VEL
LIN {X 0,Y 199.58,Z 837.747,A -85,B 0,C 180,E1 -22986.438,E2 -22986.438} C_VEL
LIN {X 0,Y 200.815,Z 824.969,A -85,B 0,C 180,E1 -22987.532,E2 -22987.532} C_VEL
LIN {X 0,Y 201.559,Z 812.021,A -85,B 0,C 180,E1 -22988.23,E2 -22988.23} C_VEL
LIN {X 0,Y 202.519,Z 781.675,A -85,B 0,C 180,E1 -22989.38,E2 -22989.38} C_VEL
LIN {X 0,Y 195.485,Z 767.899,A -85,B 0,C 180,E1 -22991.827,E2 -22991.827} C_VEL
LIN {X 0,Y 188.759,Z 756.47,A -85,B 0,C 180,E1 -22994.351,E2 -22994.351} C_VEL
LIN {X 0,Y 181.223,Z 745.207,A -85,B 0,C 180,E1 -22997.471,E2 -22997.471} C_VEL
LIN {X 0,Y 178.634,Z 741.536,A -85,B 0,C 180,E1 -22998.639,E2 -22998.639} C_VEL
LIN {X 0,Y 175.825,Z 738.105,A -85,B 0,C 180,E1 -22999.945,E2 -22999.945} C_VEL
LIN {X 0,Y 174.915,Z 736.404,A -85,B 0,C 180,E1 -23000.423,E2 -23000.423} C_VEL
LIN {X 0,Y 172.627,Z 734.323,A -85,B 0,C 180,E1 -23001.523,E2 -23001.523} C_VEL
LIN {X 0,Y 171.53,Z 731.88,A -85,B 0,C 180,E1 -23002.171,E2 -23002.171} C_VEL
LIN {X 0,Y 171.393,Z 731.13,A -85,B 0,C 180,E1 -23002.321,E2 -23002.321} C_VEL
LIN {X 0,Y 171.37,Z 731.136,A -85,B 0,C 180,E1 -23007.782,E2 -23007.782} C_VEL
LIN {X 0,Y 171.397,Z 731.119,A -85,B 0,C 180,E1 -23010.524,E2 -23010.524} C_VEL
LIN {X 0,Y 171.392,Z 731.12,A -85,B 0,C 180,E1 -23015.792,E2 -23015.792} C_VEL
LIN {X 0,Y 171.523,Z 731.109,A -85,B 0,C 180,E1 -23020.865,E2 -23020.865} C_VEL
LIN {X 0,Y 171.517,Z 731.122,A -85,B 0,C 180,E1 -23025.768,E2 -23025.768} C_VEL
LIN {X 0,Y 171.804,Z 731.071,A -85,B 0,C 180,E1 -23030.582,E2 -23030.582} C_VEL
LIN {X 0,Y 171.769,Z 731.074,A -85,B 0,C 180,E1 -23035.306,E2 -23035.306} C_VEL
LIN {X 0,Y 172.278,Z 731.031,A -85,B 0,C 180,E1 -23040,E2 -23040} C_VEL
LIN {X 0,Y 171.77,Z 731.085,A -85,B 0,C 180,E1 -23044.694,E2 -23044.694} C_VEL
LIN {X 0,Y 171.804,Z 731.068,A -85,B 0,C 180,E1 -23049.417,E2 -23049.417} C_VEL
LIN {X 0,Y 171.517,Z 731.118,A -85,B 0,C 180,E1 -23054.232,E2 -23054.232} C_VEL
LIN {X 0,Y 171.487,Z 731.111,A -85,B 0,C 180,E1 -23059.564,E2 -23059.564} C_VEL
LIN {X 0,Y 171.406,Z 731.118,A -85,B 0,C 180,E1 -23065.616,E2 -23065.616} C_VEL
LIN {X 0,Y 171.385,Z 731.262,A -85,B 0,C 180,E1 -23067.639,E2 -23067.639} C_VEL
LIN {X 0,Y 173.77,Z 738.403,A -85,B 0,C 180,E1 -23073.093,E2 -23073.093} C_VEL
LIN {X 0,Y 175.883,Z 745.068,A -85,B 0,C 180,E1 -23077.544,E2 -23077.544} C_VEL
LIN {X 0,Y 176.729,Z 747.74,A -85,B 0,C 180,E1 -23079.055,E2 -23079.055} C_VEL
LIN {X 0,Y 179.624,Z 753.001,A -85,B 0,C 180,E1 -23080.454,E2 -23080.454} C_VEL
LIN {X 0,Y 181.282,Z 756.189,A -85,B 0,C 180,E1 -23081.228,E2 -23081.228} C_VEL
LIN {X 0,Y 184.218,Z 761.666,A -85,B 0,C 180,E1 -23082.53,E2 -23082.53} C_VEL
LIN {X 0,Y 189.436,Z 772.416,A -85,B 0,C 180,E1 -23084.729,E2 -23084.729} C_VEL
LIN {X 0,Y 195.167,Z 785.979,A -85,B 0,C 180,E1 -23087.009,E2 -23087.009} C_VEL
LIN {X 0,Y 195.796,Z 788.23,A -85,B 0,C 180,E1 -23087.283,E2 -23087.283} C_VEL
LIN {X 0,Y 197.845,Z 812.882,A -85,B 0,C 180,E1 -23088.965,E2 -23088.965} C_VEL
LIN {X 0,Y 199.424,Z 842.619,A -85,B 0,C 180,E1 -23090.695,E2 -23090.695} C_VEL
LIN {X 0,Y 198.205,Z 864.202,A -85,B 0,C 180,E1 -23091.494,E2 -23091.494} C_VEL
LIN {X 0,Y 197.088,Z 873.961,A -85,B 0,C 180,E1 -23092.058,E2 -23092.058} C_VEL
LIN {X 0,Y 196.126,Z 877.726,A -85,B 0,C 180,E1 -23092.247,E2 -23092.247} C_VEL
LIN {X 0,Y 193.119,Z 884.996,A -85,B 0,C 180,E1 -23092.518,E2 -23092.518} C_VEL
LIN {X 0,Y 187.795,Z 895.494,A -85,B 0,C 180,E1 -23093.089,E2 -23093.089} C_VEL
LIN {X 0,Y 185.639,Z 900.714,A -85,B 0,C 180,E1 -23093.647,E2 -23093.647} C_VEL
LIN {X 0,Y 185.091,Z 902.402,A -85,B 0,C 180,E1 -23093.886,E2 -23093.886} C_VEL
LIN {X 0,Y 181.445,Z 913.786,A -85,B 0,C 180,E1 -23095.852,E2 -23095.852} C_VEL
LIN {X 0,Y 177.327,Z 924.731,A -85,B 0,C 180,E1 -23098.343,E2 -23098.343} C_VEL
LIN {X 0,Y 173.777,Z 933.68,A -85,B 0,C 180,E1 -23100.987,E2 -23100.987} C_VEL
LIN {X 0,Y 170.136,Z 942.45,A -85,B 0,C 180,E1 -23104.314,E2 -23104.314} C_VEL
LIN {X 0,Y 167.281,Z 949.529,A -85,B 0,C 180,E1 -23107.802,E2 -23107.802} C_VEL
LIN {X 0,Y 165.191,Z 955.258,A -85,B 0,C 180,E1 -23111.411,E2 -23111.411} C_VEL
LIN {X 0,Y 163.843,Z 959.814,A -85,B 0,C 180,E1 -23115.104,E2 -23115.104} C_VEL
LIN {X 0,Y 163.228,Z 963.312,A -85,B 0,C 180,E1 -23118.846,E2 -23118.846} C_VEL
LIN {X 0,Y 163.315,Z 965.831,A -85,B 0,C 180,E1 -23122.599,E2 -23122.599} C_VEL
LIN {X 0,Y 163.612,Z 966.964,A -85,B 0,C 180,E1 -23125.088,E2 -23125.088} C_VEL
LIN {X 0,Y 163.979,Z 967.678,A -85,B 0,C 180,E1 -23127.56,E2 -23127.56} C_VEL
LIN {X 0,Y 164.377,Z 967.961,A -85,B 0,C 180,E1 -23130.016,E2 -23130.016} C_VEL
LIN {X 0,Y 163.959,Z 967.655,A -85,B 0,C 180,E1 -23132.473,E2 -23132.473} C_VEL
LIN {X 0,Y 163.59,Z 966.926,A -85,B 0,C 180,E1 -23134.945,E2 -23134.945} C_VEL
LIN {X 0,Y 163.287,Z 965.391,A -85,B 0,C 180,E1 -23138.135,E2 -23138.135} C_VEL
LIN {X 0,Y 163.558,Z 962.202,A -85,B 0,C 180,E1 -23142.422,E2 -23142.422} C_VEL
LIN {X 0,Y 165.115,Z 957.263,A -85,B 0,C 180,E1 -23147.031,E2 -23147.031} C_VEL
LIN {X 0,Y 165.281,Z 957.009,A -85,B 0,C 180,E1 -23147.332,E2 -23147.332} C_VEL
LIN {X 0,Y 167.632,Z 956.451,A -85,B 0,C 180,E1 -23152.184,E2 -23152.184} C_VEL
LIN {X 0,Y 171.818,Z 954.737,A -85,B 0,C 180,E1 -23156.755,E2 -23156.755} C_VEL
LIN {X 0,Y 177.427,Z 951.782,A -85,B 0,C 180,E1 -23161.009,E2 -23161.009} C_VEL
LIN {X 0,Y 182.527,Z 948.872,A -85,B 0,C 180,E1 -23163.954,E2 -23163.954} C_VEL
LIN {X 0,Y 188.443,Z 945.307,A -85,B 0,C 180,E1 -23166.65,E2 -23166.65} C_VEL
LIN {X 0,Y 197.304,Z 939.271,A -85,B 0,C 180,E1 -23169.893,E2 -23169.893} C_VEL
LIN {X 0,Y 205.937,Z 932.774,A -85,B 0,C 180,E1 -23172.391,E2 -23172.391} C_VEL
LIN {X 0,Y 215.29,Z 924.935,A -85,B 0,C 180,E1 -23174.589,E2 -23174.589} C_VEL
LIN {X 0,Y 223.936,Z 917.028,A -85,B 0,C 180,E1 -23176.219,E2 -23176.219} C_VEL
LIN {X 0,Y 232.95,Z 907.744,A -85,B 0,C 180,E1 -23177.672,E2 -23177.672} C_VEL
LIN {X 0,Y 233.798,Z 906.814,A -85,B 0,C 180,E1 -23177.797,E2 -23177.797} C_VEL
LIN {X 0,Y 234.081,Z 906.277,A -85,B 0,C 180,E1 -23178.261,E2 -23178.261} C_VEL
LIN {X 0,Y 228.029,Z 911.398,A -85,B 0,C 180,E1 -23179.666,E2 -23179.666} C_VEL
LIN {X 0,Y 220.546,Z 916.923,A -85,B 0,C 180,E1 -23181.582,E2 -23181.582} C_VEL
LIN {X 0,Y 213.371,Z 921.371,A -85,B 0,C 180,E1 -23183.638,E2 -23183.638} C_VEL
LIN {X 0,Y 208.821,Z 923.814,A -85,B 0,C 180,E1 -23185.1,E2 -23185.1} C_VEL
LIN {X 0,Y 200.141,Z 927.345,A -85,B 0,C 180,E1 -23188.215,E2 -23188.215} C_VEL
LIN {X 0,Y 196.079,Z 928.618,A -85,B 0,C 180,E1 -23189.881,E2 -23189.881} C_VEL
LIN {X 0,Y 188.516,Z 929.833,A -85,B 0,C 180,E1 -23193.425,E2 -23193.425} C_VEL
LIN {X 0,Y 181.861,Z 929.678,A -85,B 0,C 180,E1 -23197.266,E2 -23197.266} C_VEL
LIN {X 0,Y 176.137,Z 927.924,A -85,B 0,C 180,E1 -23201.385,E2 -23201.385} C_VEL
LIN {X 0,Y 171.47,Z 924.672,A -85,B 0,C 180,E1 -23205.764,E2 -23205.764} C_VEL
LIN {X 0,Y 168.155,Z 919.737,A -85,B 0,C 180,E1 -23210.376,E2 -23210.376} C_VEL
LIN {X 0,Y 166.336,Z 914.945,A -85,B 0,C 180,E1 -23213.937,E2 -23213.937} C_VEL
LIN {X 0,Y 165.011,Z 909.085,A -85,B 0,C 180,E1 -23217.559,E2 -23217.559} C_VEL
LIN {X 0,Y 164.32,Z 901.952,A -85,B 0,C 180,E1 -23221.226,E2 -23221.226} C_VEL
LIN {X 0,Y 164.164,Z 894.931,A -85,B 0,C 180,E1 -23224.297,E2 -23224.297} C_VEL
LIN {X 0,Y 164.529,Z 886.776,A -85,B 0,C 180,E1 -23227.363,E2 -23227.363} C_VEL
LIN {X 0,Y 165.024,Z 877.579,A -85,B 0,C 180,E1 -23230.262,E2 -23230.262} C_VEL
LIN {X 0,Y 165.719,Z 867.838,A -85,B 0,C 180,E1 -23232.864,E2 -23232.864} C_VEL
LIN {X 0,Y 166.609,Z 855.549,A -85,B 0,C 180,E1 -23235.6,E2 -23235.6} C_VEL
LIN {X 0,Y 167.604,Z 841.663,A -85,B 0,C 180,E1 -23238.014,E2 -23238.014} C_VEL
LIN {X 0,Y 168.281,Z 830.721,A -85,B 0,C 180,E1 -23239.519,E2 -23239.519} C_VEL
LIN {X 0,Y 168.893,Z 818.947,A -85,B 0,C 180,E1 -23240.794,E2 -23240.794} C_VEL
LIN {X 0,Y 169.529,Z 801.307,A -85,B 0,C 180,E1 -23242.228,E2 -23242.228} C_VEL
LIN {X 0,Y 171.071,Z 757.219,A -85,B 0,C 180,E1 -23245.529,E2 -23245.529} C_VEL
LIN {X 0,Y 164.527,Z 731.987,A -85,B 0,C 180,E1 -23247.745,E2 -23247.745} C_VEL
LIN {X 0,Y 164.353,Z 732.008,A -85,B 0,C 180,E1 -23253.773,E2 -23253.773} C_VEL
LIN {X 0,Y 164.396,Z 732.041,A -85,B 0,C 180,E1 -23254.642,E2 -23254.642} C_VEL
LIN {X 0,Y 165.267,Z 734.681,A -85,B 0,C 180,E1 -23255.294,E2 -23255.294} C_VEL
LIN {X 0,Y 167.212,Z 736.861,A -85,B 0,C 180,E1 -23256.419,E2 -23256.419} C_VEL
LIN {X 0,Y 168.278,Z 737.746,A -85,B 0,C 180,E1 -23256.99,E2 -23256.99} C_VEL
LIN {X 0,Y 170.313,Z 741.031,A -85,B 0,C 180,E1 -23258.148,E2 -23258.148} C_VEL
LIN {X 0,Y 172.01,Z 742.86,A -85,B 0,C 180,E1 -23259.01,E2 -23259.01} C_VEL
LIN {X 0,Y 174.68,Z 746.568,A -85,B 0,C 180,E1 -23260.355,E2 -23260.355} C_VEL
LIN {X 0,Y 179.05,Z 752.84,A -85,B 0,C 180,E1 -23262.406,E2 -23262.406} C_VEL
LIN {X 0,Y 185.515,Z 762.72,A -85,B 0,C 180,E1 -23265.165,E2 -23265.165} C_VEL
LIN {X 0,Y 191.823,Z 773.748,A -85,B 0,C 180,E1 -23267.633,E2 -23267.633} C_VEL
LIN {X 0,Y 196.904,Z 783.995,A -85,B 0,C 180,E1 -23269.506,E2 -23269.506} C_VEL
LIN {X 0,Y 195.598,Z 819.674,A -85,B 0,C 180,E1 -23270.957,E2 -23270.957} C_VEL
LIN {X 0,Y 194.51,Z 832.708,A -85,B 0,C 180,E1 -23271.886,E2 -23271.886} C_VEL
LIN {X 0,Y 192.583,Z 845.383,A -85,B 0,C 180,E1 -23273.143,E2 -23273.143} C_VEL
LIN {X 0,Y 190.222,Z 856.749,A -85,B 0,C 180,E1 -23274.683,E2 -23274.683} C_VEL
LIN {X 0,Y 187.17,Z 868.176,A -85,B 0,C 180,E1 -23276.677,E2 -23276.677} C_VEL
LIN {X 0,Y 184.064,Z 878.261,A -85,B 0,C 180,E1 -23278.957,E2 -23278.957} C_VEL
LIN {X 0,Y 180.9,Z 887.285,A -85,B 0,C 180,E1 -23281.566,E2 -23281.566} C_VEL
LIN {X 0,Y 177.278,Z 896.06,A -85,B 0,C 180,E1 -23284.76,E2 -23284.76} C_VEL
LIN {X 0,Y 173.856,Z 903.721,A -85,B 0,C 180,E1 -23288.398,E2 -23288.398} C_VEL
LIN {X 0,Y 171.289,Z 909.479,A -85,B 0,C 180,E1 -23292.063,E2 -23292.063} C_VEL
LIN {X 0,Y 169.884,Z 912.412,A -85,B 0,C 180,E1 -23294.386,E2 -23294.386} C_VEL
LIN {X 0,Y 167.802,Z 915.967,A -85,B 0,C 180,E1 -23297.897,E2 -23297.897} C_VEL
LIN {X 0,Y 166.817,Z 917.788,A -85,B 0,C 180,E1 -23300.283,E2 -23300.283} C_VEL
LIN {X 0,Y 165.802,Z 920.09,A -85,B 0,C 180,E1 -23305.121,E2 -23305.121} C_VEL
LIN {X 0,Y 165.307,Z 920.925,A -85,B 0,C 180,E1 -23309.984,E2 -23309.984} C_VEL
LIN {X 0,Y 165.793,Z 920.154,A -85,B 0,C 180,E1 -23314.847,E2 -23314.847} C_VEL
LIN {X 0,Y 166.787,Z 917.92,A -85,B 0,C 180,E1 -23319.687,E2 -23319.687} C_VEL
LIN {X 0,Y 168.393,Z 915.094,A -85,B 0,C 180,E1 -23323.253,E2 -23323.253} C_VEL
LIN {X 0,Y 170.486,Z 911.262,A -85,B 0,C 180,E1 -23326.754,E2 -23326.754} C_VEL
LIN {X 0,Y 173.032,Z 905.781,A -85,B 0,C 180,E1 -23330.564,E2 -23330.564} C_VEL
LIN {X 0,Y 176.143,Z 898.96,A -85,B 0,C 180,E1 -23334.122,E2 -23334.122} C_VEL
LIN {X 0,Y 179.596,Z 890.923,A -85,B 0,C 180,E1 -23337.356,E2 -23337.356} C_VEL
LIN {X 0,Y 182.697,Z 882.692,A -85,B 0,C 180,E1 -23339.986,E2 -23339.986} C_VEL
LIN {X 0,Y 186.044,Z 872.503,A -85,B 0,C 180,E1 -23342.549,E2 -23342.549} C_VEL
LIN {X 0,Y 189.095,Z 862.018,A -85,B 0,C 180,E1 -23344.59,E2 -23344.59} C_VEL
LIN {X 0,Y 191.764,Z 850.725,A -85,B 0,C 180,E1 -23346.311,E2 -23346.311} C_VEL
LIN {X 0,Y 193.975,Z 838.741,A -85,B 0,C 180,E1 -23347.671,E2 -23347.671} C_VEL
LIN {X 0,Y 195.321,Z 825.718,A -85,B 0,C 180,E1 -23348.802,E2 -23348.802} C_VEL
LIN {X 0,Y 196.089,Z 812.725,A -85,B 0,C 180,E1 -23349.514,E2 -23349.514} C_VEL
LIN {X 0,Y 197.133,Z 784.24,A -85,B 0,C 180,E1 -23350.601,E2 -23350.601} C_VEL
LIN {X 0,Y 190.073,Z 770.393,A -85,B 0,C 180,E1 -23353.229,E2 -23353.229} C_VEL
LIN {X 0,Y 182.882,Z 758.357,A -85,B 0,C 180,E1 -23356.139,E2 -23356.139} C_VEL
LIN {X 0,Y 177.277,Z 750.13,A -85,B 0,C 180,E1 -23358.629,E2 -23358.629} C_VEL
LIN {X 0,Y 174.478,Z 746.266,A -85,B 0,C 180,E1 -23359.968,E2 -23359.968} C_VEL
LIN {X 0,Y 171.497,Z 742.136,A -85,B 0,C 180,E1 -23361.489,E2 -23361.489} C_VEL
LIN {X 0,Y 169.107,Z 739.294,A -85,B 0,C 180,E1 -23362.756,E2 -23362.756} C_VEL
LIN {X 0,Y 168.008,Z 737.355,A -85,B 0,C 180,E1 -23363.409,E2 -23363.409} C_VEL
LIN {X 0,Y 165.683,Z 735.353,A -85,B 0,C 180,E1 -23364.698,E2 -23364.698} C_VEL
LIN {X 0,Y 164.465,Z 732.876,A -85,B 0,C 180,E1 -23365.516,E2 -23365.516} C_VEL
LIN {X 0,Y 164.304,Z 732.005,A -85,B 0,C 180,E1 -23365.689,E2 -23365.689} C_VEL
LIN {X 0,Y 164.34,Z 732.008,A -85,B 0,C 180,E1 -23369.124,E2 -23369.124} C_VEL
LIN {X 0,Y 164.354,Z 732.005,A -85,B 0,C 180,E1 -23374.684,E2 -23374.684} C_VEL
LIN {X 0,Y 164.431,Z 732.001,A -85,B 0,C 180,E1 -23380.045,E2 -23380.045} C_VEL
LIN {X 0,Y 164.447,Z 731.998,A -85,B 0,C 180,E1 -23385.142,E2 -23385.142} C_VEL
LIN {X 0,Y 164.73,Z 731.949,A -85,B 0,C 180,E1 -23390.174,E2 -23390.174} C_VEL
LIN {X 0,Y 164.781,Z 731.965,A -85,B 0,C 180,E1 -23392.649,E2 -23392.649} C_VEL
LIN {X 0,Y 165.003,Z 731.921,A -85,B 0,C 180,E1 -23397.559,E2 -23397.559} C_VEL
LIN {X 0,Y 165.241,Z 731.908,A -85,B 0,C 180,E1 -23400,E2 -23400} C_VEL
LIN {X 0,Y 164.718,Z 731.965,A -85,B 0,C 180,E1 -23404.895,E2 -23404.895} C_VEL
LIN {X 0,Y 164.781,Z 731.954,A -85,B 0,C 180,E1 -23407.351,E2 -23407.351} C_VEL
LIN {X 0,Y 164.689,Z 731.965,A -85,B 0,C 180,E1 -23411.14,E2 -23411.14} C_VEL
LIN {X 0,Y 164.425,Z 732.001,A -85,B 0,C 180,E1 -23417.41,E2 -23417.41} C_VEL
LIN {X 0,Y 164.42,Z 731.988,A -85,B 0,C 180,E1 -23419.996,E2 -23419.996} C_VEL
LIN {X 0,Y 164.376,Z 732.176,A -85,B 0,C 180,E1 -23424.974,E2 -23424.974} C_VEL
LIN {X 0,Y 166.525,Z 738.573,A -85,B 0,C 180,E1 -23430.427,E2 -23430.427} C_VEL
LIN {X 0,Y 168.724,Z 745.475,A -85,B 0,C 180,E1 -23435.489,E2 -23435.489} C_VEL
LIN {X 0,Y 172.014,Z 751.329,A -85,B 0,C 180,E1 -23437.384,E2 -23437.384} C_VEL
LIN {X 0,Y 173.493,Z 753.752,A -85,B 0,C 180,E1 -23438.153,E2 -23438.153} C_VEL
LIN {X 0,Y 176.99,Z 760.138,A -85,B 0,C 180,E1 -23439.913,E2 -23439.913} C_VEL
LIN {X 0,Y 180.693,Z 767.421,A -85,B 0,C 180,E1 -23441.671,E2 -23441.671} C_VEL
LIN {X 0,Y 185.254,Z 777.158,A -85,B 0,C 180,E1 -23443.709,E2 -23443.709} C_VEL
LIN {X 0,Y 190.615,Z 790.271,A -85,B 0,C 180,E1 -23445.982,E2 -23445.982} C_VEL
LIN {X 0,Y 192.567,Z 816.287,A -85,B 0,C 180,E1 -23447.797,E2 -23447.797} C_VEL
LIN {X 0,Y 193.905,Z 843.794,A -85,B 0,C 180,E1 -23449.45,E2 -23449.45} C_VEL
LIN {X 0,Y 192.684,Z 863.464,A -85,B 0,C 180,E1 -23450.195,E2 -23450.195} C_VEL
LIN {X 0,Y 190.966,Z 876.461,A -85,B 0,C 180,E1 -23451.002,E2 -23451.002} C_VEL
LIN {X 0,Y 188.585,Z 888.445,A -85,B 0,C 180,E1 -23452.076,E2 -23452.076} C_VEL
LIN {X 0,Y 185.437,Z 901.195,A -85,B 0,C 180,E1 -23453.709,E2 -23453.709} C_VEL
LIN {X 0,Y 185.091,Z 902.402,A -85,B 0,C 180,E1 -23453.886,E2 -23453.886} C_VEL
LIN {X 0,Y 182.976,Z 907.463,A -85,B 0,C 180,E1 -23454.576,E2 -23454.576} C_VEL
LIN {X 0,Y 177.744,Z 915.277,A -85,B 0,C 180,E1 -23455.595,E2 -23455.595} C_VEL
LIN {X 0,Y 172.337,Z 922.608,A -85,B 0,C 180,E1 -23456.88,E2 -23456.88} C_VEL
LIN {X 0,Y 169.988,Z 926.909,A -85,B 0,C 180,E1 -23457.982,E2 -23457.982} C_VEL
LIN {X 0,Y 166.176,Z 935.779,A -85,B 0,C 180,E1 -23460.919,E2 -23460.919} C_VEL
LIN {X 0,Y 162.639,Z 943.968,A -85,B 0,C 180,E1 -23464.418,E2 -23464.418} C_VEL
LIN {X 0,Y 159.822,Z 950.581,A -85,B 0,C 180,E1 -23468.071,E2 -23468.071} C_VEL
LIN {X 0,Y 157.83,Z 955.899,A -85,B 0,C 180,E1 -23471.857,E2 -23471.857} C_VEL
LIN {X 0,Y 156.591,Z 960.091,A -85,B 0,C 180,E1 -23475.728,E2 -23475.728} C_VEL
LIN {X 0,Y 156.16,Z 963.264,A -85,B 0,C 180,E1 -23479.647,E2 -23479.647} C_VEL
LIN {X 0,Y 156.227,Z 964.811,A -85,B 0,C 180,E1 -23482.262,E2 -23482.262} C_VEL
LIN {X 0,Y 156.533,Z 965.951,A -85,B 0,C 180,E1 -23484.866,E2 -23484.866} C_VEL
LIN {X 0,Y 156.902,Z 966.668,A -85,B 0,C 180,E1 -23487.45,E2 -23487.45} C_VEL
LIN {X 0,Y 157.323,Z 966.955,A -85,B 0,C 180,E1 -23490.017,E2 -23490.017} C_VEL
LIN {X 0,Y 156.883,Z 966.644,A -85,B 0,C 180,E1 -23492.584,E2 -23492.584} C_VEL
LIN {X 0,Y 156.515,Z 965.912,A -85,B 0,C 180,E1 -23495.169,E2 -23495.169} C_VEL
LIN {X 0,Y 156.222,Z 964.537,A -85,B 0,C 180,E1 -23498.222,E2 -23498.222} C_VEL
LIN {X 0,Y 156.611,Z 961.185,A -85,B 0,C 180,E1 -23502.983,E2 -23502.983} C_VEL
LIN {X 0,Y 157.865,Z 957.363,A -85,B 0,C 180,E1 -23506.837,E2 -23506.837} C_VEL
LIN {X 0,Y 158.812,Z 955.289,A -85,B 0,C 180,E1 -23508.73,E2 -23508.73} C_VEL
LIN {X 0,Y 162.272,Z 954.716,A -85,B 0,C 180,E1 -23514.562,E2 -23514.562} C_VEL
LIN {X 0,Y 165.526,Z 953.692,A -85,B 0,C 180,E1 -23517.859,E2 -23517.859} C_VEL
LIN {X 0,Y 171.379,Z 951.243,A -85,B 0,C 180,E1 -23522.232,E2 -23522.232} C_VEL
LIN {X 0,Y 178.623,Z 947.67,A -85,B 0,C 180,E1 -23526.185,E2 -23526.185} C_VEL
LIN {X 0,Y 187.259,Z 942.893,A -85,B 0,C 180,E1 -23529.66,E2 -23529.66} C_VEL
LIN {X 0,Y 196.883,Z 936.79,A -85,B 0,C 180,E1 -23532.72,E2 -23532.72} C_VEL
LIN {X 0,Y 207.558,Z 929.181,A -85,B 0,C 180,E1 -23535.336,E2 -23535.336} C_VEL
LIN {X 0,Y 216.141,Z 922.357,A -85,B 0,C 180,E1 -23537.036,E2 -23537.036} C_VEL
LIN {X 0,Y 222.444,Z 917.033,A -85,B 0,C 180,E1 -23538.084,E2 -23538.084} C_VEL
LIN {X 0,Y 223.406,Z 915.904,A -85,B 0,C 180,E1 -23538.652,E2 -23538.652} C_VEL
LIN {X 0,Y 213.138,Z 922.245,A -85,B 0,C 180,E1 -23541.207,E2 -23541.207} C_VEL
LIN {X 0,Y 205.83,Z 925.84,A -85,B 0,C 180,E1 -23543.307,E2 -23543.307} C_VEL
LIN {X 0,Y 198.906,Z 928.549,A -85,B 0,C 180,E1 -23545.574,E2 -23545.574} C_VEL
LIN {X 0,Y 190.223,Z 930.768,A -85,B 0,C 180,E1 -23548.852,E2 -23548.852} C_VEL
LIN {X 0,Y 186.216,Z 931.402,A -85,B 0,C 180,E1 -23550.618,E2 -23550.618} C_VEL
LIN {X 0,Y 178.806,Z 931.415,A -85,B 0,C 180,E1 -23554.383,E2 -23554.383} C_VEL
LIN {X 0,Y 172.295,Z 929.987,A -85,B 0,C 180,E1 -23558.462,E2 -23558.462} C_VEL
LIN {X 0,Y 166.888,Z 926.955,A -85,B 0,C 180,E1 -23562.855,E2 -23562.855} C_VEL
LIN {X 0,Y 163.649,Z 923.696,A -85,B 0,C 180,E1 -23566.338,E2 -23566.338} C_VEL
LIN {X 0,Y 160.524,Z 918.034,A -85,B 0,C 180,E1 -23571.186,E2 -23571.186} C_VEL
LIN {X 0,Y 158.557,Z 911.468,A -85,B 0,C 180,E1 -23575.551,E2 -23575.551} C_VEL
LIN {X 0,Y 157.493,Z 904.572,A -85,B 0,C 180,E1 -23579.361,E2 -23579.361} C_VEL
LIN {X 0,Y 157.142,Z 897.835,A -85,B 0,C 180,E1 -23582.563,E2 -23582.563} C_VEL
LIN {X 0,Y 157.27,Z 889.914,A -85,B 0,C 180,E1 -23585.771,E2 -23585.771} C_VEL
LIN {X 0,Y 157.79,Z 880.631,A -85,B 0,C 180,E1 -23588.969,E2 -23588.969} C_VEL
LIN {X 0,Y 158.309,Z 872.008,A -85,B 0,C 180,E1 -23591.507,E2 -23591.507} C_VEL
LIN {X 0,Y 159.006,Z 862.2,A -85,B 0,C 180,E1 -23593.939,E2 -23593.939} C_VEL
LIN {X 0,Y 159.7,Z 852.533,A -85,B 0,C 180,E1 -23595.965,E2 -23595.965} C_VEL
LIN {X 0,Y 160.556,Z 840.746,A -85,B 0,C 180,E1 -23598.008,E2 -23598.008} C_VEL
LIN {X 0,Y 161.25,Z 829.537,A -85,B 0,C 180,E1 -23599.576,E2 -23599.576} C_VEL
LIN {X 0,Y 161.96,Z 815.893,A -85,B 0,C 180,E1 -23601.061,E2 -23601.061} C_VEL
LIN {X 0,Y 163.949,Z 758.096,A -85,B 0,C 180,E1 -23605.671,E2 -23605.671} C_VEL
LIN {X 0,Y 157.476,Z 732.865,A -85,B 0,C 180,E1 -23607.998,E2 -23607.998} C_VEL
LIN {X 0,Y 157.377,Z 732.999,A -85,B 0,C 180,E1 -23610.665,E2 -23610.665} C_VEL
LIN {X 0,Y 158.185,Z 735.476,A -85,B 0,C 180,E1 -23611.394,E2 -23611.394} C_VEL
LIN {X 0,Y 160.086,Z 737.681,A -85,B 0,C 180,E1 -23612.721,E2 -23612.721} C_VEL
LIN {X 0,Y 161.604,Z 738.841,A -85,B 0,C 180,E1 -23613.676,E2 -23613.676} C_VEL
LIN {X 0,Y 163.344,Z 741.795,A -85,B 0,C 180,E1 -23614.845,E2 -23614.845} C_VEL
LIN {X 0,Y 165.443,Z 743.964,A -85,B 0,C 180,E1 -23616.077,E2 -23616.077} C_VEL
LIN {X 0,Y 168.088,Z 747.67,A -85,B 0,C 180,E1 -23617.603,E2 -23617.603} C_VEL
LIN {X 0,Y 169.673,Z 749.899,A -85,B 0,C 180,E1 -23618.471,E2 -23618.471} C_VEL
LIN {X 0,Y 172.842,Z 754.312,A -85,B 0,C 180,E1 -23620.108,E2 -23620.108} C_VEL
LIN {X 0,Y 177.341,Z 760.887,A -85,B 0,C 180,E1 -23622.262,E2 -23622.262} C_VEL
LIN {X 0,Y 183.704,Z 771.283,A -85,B 0,C 180,E1 -23625.053,E2 -23625.053} C_VEL
LIN {X 0,Y 189.443,Z 782.191,A -85,B 0,C 180,E1 -23627.384,E2 -23627.384} C_VEL
LIN {X 0,Y 191.578,Z 786.567,A -85,B 0,C 180,E1 -23628.209,E2 -23628.209} C_VEL
LIN {X 0,Y 190.205,Z 820.579,A -85,B 0,C 180,E1 -23629.618,E2 -23629.618} C_VEL
LIN {X 0,Y 189.088,Z 833.26,A -85,B 0,C 180,E1 -23630.533,E2 -23630.533} C_VEL
LIN {X 0,Y 187.241,Z 845.205,A -85,B 0,C 180,E1 -23631.72,E2 -23631.72} C_VEL
LIN {X 0,Y 184.824,Z 856.613,A -85,B 0,C 180,E1 -23633.24,E2 -23633.24} C_VEL
LIN {X 0,Y 181.725,Z 867.912,A -85,B 0,C 180,E1 -23635.204,E2 -23635.204} C_VEL
LIN {X 0,Y 178.435,Z 878.222,A -85,B 0,C 180,E1 -23637.529,E2 -23637.529} C_VEL
LIN {X 0,Y 175.415,Z 886.621,A -85,B 0,C 180,E1 -23639.931,E2 -23639.931} C_VEL
LIN {X 0,Y 172.173,Z 894.37,A -85,B 0,C 180,E1 -23642.648,E2 -23642.648} C_VEL
LIN {X 0,Y 168.661,Z 902.038,A -85,B 0,C 180,E1 -23646.079,E2 -23646.079} C_VEL
LIN {X 0,Y 165.989,Z 907.665,A -85,B 0,C 180,E1 -23649.326,E2 -23649.326} C_VEL
LIN {X 0,Y 163.126,Z 913.416,A -85,B 0,C 180,E1 -23653.721,E2 -23653.721} C_VEL
LIN {X 0,Y 160.937,Z 916.97,A -85,B 0,C 180,E1 -23657.372,E2 -23657.372} C_VEL
LIN {X 0,Y 159.893,Z 918.791,A -85,B 0,C 180,E1 -23659.858,E2 -23659.858} C_VEL
LIN {X 0,Y 158.8,Z 921.093,A -85,B 0,C 180,E1 -23664.905,E2 -23664.905} C_VEL
LIN {X 0,Y 158.279,Z 921.927,A -85,B 0,C 180,E1 -23669.983,E2 -23669.983} C_VEL
LIN {X 0,Y 158.791,Z 921.157,A -85,B 0,C 180,E1 -23675.061,E2 -23675.061} C_VEL
LIN {X 0,Y 159.863,Z 918.922,A -85,B 0,C 180,E1 -23680.11,E2 -23680.11} C_VEL
LIN {X 0,Y 161.561,Z 916.096,A -85,B 0,C 180,E1 -23683.824,E2 -23683.824} C_VEL
LIN {X 0,Y 163.769,Z 912.264,A -85,B 0,C 180,E1 -23687.463,E2 -23687.463} C_VEL
LIN {X 0,Y 166.47,Z 906.782,A -85,B 0,C 180,E1 -23691.414,E2 -23691.414} C_VEL
LIN {X 0,Y 169.753,Z 899.961,A -85,B 0,C 180,E1 -23695.091,E2 -23695.091} C_VEL
LIN {X 0,Y 173.384,Z 891.923,A -85,B 0,C 180,E1 -23698.423,E2 -23698.423} C_VEL
LIN {X 0,Y 176.647,Z 883.691,A -85,B 0,C 180,E1 -23701.125,E2 -23701.125} C_VEL
LIN {X 0,Y 180.159,Z 873.501,A -85,B 0,C 180,E1 -23703.752,E2 -23703.752} C_VEL
LIN {X 0,Y 183.358,Z 863.015,A -85,B 0,C 180,E1 -23705.836,E2 -23705.836} C_VEL
LIN {X 0,Y 186.273,Z 851.186,A -85,B 0,C 180,E1 -23707.663,E2 -23707.663} C_VEL
LIN {X 0,Y 188.58,Z 838.585,A -85,B 0,C 180,E1 -23709.102,E2 -23709.102} C_VEL
LIN {X 0,Y 189.982,Z 825.719,A -85,B 0,C 180,E1 -23710.204,E2 -23710.204} C_VEL
LIN {X 0,Y 190.765,Z 812.492,A -85,B 0,C 180,E1 -23710.906,E2 -23710.906} C_VEL
LIN {X 0,Y 191.732,Z 786.736,A -85,B 0,C 180,E1 -23711.924,E2 -23711.924} C_VEL
LIN {X 0,Y 185.433,Z 774.268,A -85,B 0,C 180,E1 -23714.43,E2 -23714.43} C_VEL
LIN {X 0,Y 178.971,Z 763.299,A -85,B 0,C 180,E1 -23717.213,E2 -23717.213} C_VEL
LIN {X 0,Y 173.507,Z 755.075,A -85,B 0,C 180,E1 -23719.797,E2 -23719.797} C_VEL
LIN {X 0,Y 170.882,Z 751.46,A -85,B 0,C 180,E1 -23721.129,E2 -23721.129} C_VEL
LIN {X 0,Y 168.346,Z 747.874,A -85,B 0,C 180,E1 -23722.503,E2 -23722.503} C_VEL
LIN {X 0,Y 165.653,Z 744.27,A -85,B 0,C 180,E1 -23724.047,E2 -23724.047} C_VEL
LIN {X 0,Y 164.89,Z 743.276,A -85,B 0,C 180,E1 -23724.502,E2 -23724.502} C_VEL
LIN {X 0,Y 162.582,Z 740.762,A -85,B 0,C 180,E1 -23725.902,E2 -23725.902} C_VEL
LIN {X 0,Y 161.277,Z 738.447,A -85,B 0,C 180,E1 -23726.808,E2 -23726.808} C_VEL
LIN {X 0,Y 158.845,Z 736.558,A -85,B 0,C 180,E1 -23728.393,E2 -23728.393} C_VEL
LIN {X 0,Y 157.47,Z 733.883,A -85,B 0,C 180,E1 -23729.491,E2 -23729.491} C_VEL
LIN {X 0,Y 157.258,Z 732.883,A -85,B 0,C 180,E1 -23729.816,E2 -23729.816} C_VEL
LIN {X 0,Y 157.263,Z 732.895,A -85,B 0,C 180,E1 -23733.455,E2 -23733.455} C_VEL
LIN {X 0,Y 157.34,Z 732.887,A -85,B 0,C 180,E1 -23739.662,E2 -23739.662} C_VEL
LIN {X 0,Y 157.384,Z 732.869,A -85,B 0,C 180,E1 -23744.459,E2 -23744.459} C_VEL
LIN {X 0,Y 157.661,Z 732.827,A -85,B 0,C 180,E1 -23749.729,E2 -23749.729} C_VEL
LIN {X 0,Y 157.738,Z 732.841,A -85,B 0,C 180,E1 -23752.318,E2 -23752.318} C_VEL
LIN {X 0,Y 157.951,Z 732.798,A -85,B 0,C 180,E1 -23757.45,E2 -23757.45} C_VEL
LIN {X 0,Y 158.203,Z 732.784,A -85,B 0,C 180,E1 -23760,E2 -23760} C_VEL
LIN {X 0,Y 157.667,Z 732.845,A -85,B 0,C 180,E1 -23765.115,E2 -23765.115} C_VEL
LIN {X 0,Y 157.719,Z 732.829,A -85,B 0,C 180,E1 -23767.682,E2 -23767.682} C_VEL
LIN {X 0,Y 157.618,Z 732.847,A -85,B 0,C 180,E1 -23771.308,E2 -23771.308} C_VEL
LIN {X 0,Y 157.395,Z 732.879,A -85,B 0,C 180,E1 -23775.54,E2 -23775.54} C_VEL
LIN {X 0,Y 157.315,Z 732.87,A -85,B 0,C 180,E1 -23780.94,E2 -23780.94} C_VEL
LIN {X 0,Y 157.271,Z 732.878,A -85,B 0,C 180,E1 -23781.634,E2 -23781.634} C_VEL
LIN {X 0,Y 158.83,Z 737.565,A -85,B 0,C 180,E1 -23786.262,E2 -23786.262} C_VEL
LIN {X 0,Y 160.418,Z 742.124,A -85,B 0,C 180,E1 -23790.253,E2 -23790.253} C_VEL
LIN {X 0,Y 161.085,Z 743.931,A -85,B 0,C 180,E1 -23791.571,E2 -23791.571} C_VEL
LIN {X 0,Y 164.262,Z 749.402,A -85,B 0,C 180,E1 -23793.682,E2 -23793.682} C_VEL
LIN {X 0,Y 165.82,Z 751.757,A -85,B 0,C 180,E1 -23794.625,E2 -23794.625} C_VEL
LIN {X 0,Y 170.067,Z 759.145,A -85,B 0,C 180,E1 -23797.075,E2 -23797.075} C_VEL
LIN {X 0,Y 173.475,Z 765.571,A -85,B 0,C 180,E1 -23798.899,E2 -23798.899} C_VEL
LIN {X 0,Y 178.12,Z 774.93,A -85,B 0,C 180,E1 -23801.208,E2 -23801.208} C_VEL
LIN {X 0,Y 182.904,Z 786.151,A -85,B 0,C 180,E1 -23803.456,E2 -23803.456} C_VEL
LIN {X 0,Y 185.613,Z 793.195,A -85,B 0,C 180,E1 -23804.677,E2 -23804.677} C_VEL
LIN {X 0,Y 187.348,Z 819.029,A -85,B 0,C 180,E1 -23806.523,E2 -23806.523} C_VEL
LIN {X 0,Y 188.406,Z 845.305,A -85,B 0,C 180,E1 -23808.128,E2 -23808.128} C_VEL
LIN {X 0,Y 187.119,Z 863.886,A -85,B 0,C 180,E1 -23808.871,E2 -23808.871} C_VEL
LIN {X 0,Y 185.248,Z 876.818,A -85,B 0,C 180,E1 -23809.72,E2 -23809.72} C_VEL
LIN {X 0,Y 182.524,Z 889.443,A -85,B 0,C 180,E1 -23810.934,E2 -23810.934} C_VEL
LIN {X 0,Y 179.268,Z 901.776,A -85,B 0,C 180,E1 -23812.601,E2 -23812.601} C_VEL
LIN {X 0,Y 175.533,Z 912.763,A -85,B 0,C 180,E1 -23814.532,E2 -23814.532} C_VEL
LIN {X 0,Y 171.325,Z 923.721,A -85,B 0,C 180,E1 -23817.097,E2 -23817.097} C_VEL
LIN {X 0,Y 169.988,Z 926.909,A -85,B 0,C 180,E1 -23817.982,E2 -23817.982} C_VEL
LIN {X 0,Y 167.656,Z 931.082,A -85,B 0,C 180,E1 -23819.187,E2 -23819.187} C_VEL
LIN {X 0,Y 162.226,Z 937.299,A -85,B 0,C 180,E1 -23821.103,E2 -23821.103} C_VEL
LIN {X 0,Y 156.905,Z 942.891,A -85,B 0,C 180,E1 -23823.321,E2 -23823.321} C_VEL
LIN {X 0,Y 154.799,Z 946.067,A -85,B 0,C 180,E1 -23824.969,E2 -23824.969} C_VEL
LIN {X 0,Y 152.381,Z 951.45,A -85,B 0,C 180,E1 -23828.368,E2 -23828.368} C_VEL
LIN {X 0,Y 150.485,Z 956.385,A -85,B 0,C 180,E1 -23832.348,E2 -23832.348} C_VEL
LIN {X 0,Y 149.373,Z 960.22,A -85,B 0,C 180,E1 -23836.413,E2 -23836.413} C_VEL
LIN {X 0,Y 149.095,Z 962.239,A -85,B 0,C 180,E1 -23839.151,E2 -23839.151} C_VEL
LIN {X 0,Y 149.168,Z 963.795,A -85,B 0,C 180,E1 -23841.893,E2 -23841.893} C_VEL
LIN {X 0,Y 149.453,Z 964.937,A -85,B 0,C 180,E1 -23844.622,E2 -23844.622} C_VEL
LIN {X 0,Y 149.826,Z 965.657,A -85,B 0,C 180,E1 -23847.329,E2 -23847.329} C_VEL
LIN {X 0,Y 150.266,Z 965.948,A -85,B 0,C 180,E1 -23850.018,E2 -23850.018} C_VEL
LIN {X 0,Y 149.808,Z 965.633,A -85,B 0,C 180,E1 -23852.707,E2 -23852.707} C_VEL
LIN {X 0,Y 149.441,Z 964.898,A -85,B 0,C 180,E1 -23855.415,E2 -23855.415} C_VEL
LIN {X 0,Y 149.181,Z 963.634,A -85,B 0,C 180,E1 -23858.38,E2 -23858.38} C_VEL
LIN {X 0,Y 149.399,Z 961.217,A -85,B 0,C 180,E1 -23862.239,E2 -23862.239} C_VEL
LIN {X 0,Y 150.5,Z 957.73,A -85,B 0,C 180,E1 -23866.289,E2 -23866.289} C_VEL
LIN {X 0,Y 152.511,Z 953.398,A -85,B 0,C 180,E1 -23870.236,E2 -23870.236} C_VEL
LIN {X 0,Y 156.877,Z 953.084,A -85,B 0,C 180,E1 -23876.632,E2 -23876.632} C_VEL
LIN {X 0,Y 162.215,Z 951.605,A -85,B 0,C 180,E1 -23881.342,E2 -23881.342} C_VEL
LIN {X 0,Y 169.058,Z 949.052,A -85,B 0,C 180,E1 -23885.608,E2 -23885.608} C_VEL
LIN {X 0,Y 177.255,Z 945.404,A -85,B 0,C 180,E1 -23889.391,E2 -23889.391} C_VEL
LIN {X 0,Y 186.672,Z 940.572,A -85,B 0,C 180,E1 -23892.678,E2 -23892.678} C_VEL
LIN {X 0,Y 197.106,Z 934.433,A -85,B 0,C 180,E1 -23895.504,E2 -23895.504} C_VEL
LIN {X 0,Y 206.973,Z 927.862,A -85,B 0,C 180,E1 -23897.622,E2 -23897.622} C_VEL
LIN {X 0,Y 213.427,Z 923.225,A -85,B 0,C 180,E1 -23898.808,E2 -23898.808} C_VEL
LIN {X 0,Y 205.628,Z 926.982,A -85,B 0,C 180,E1 -23900.78,E2 -23900.78} C_VEL
LIN {X 0,Y 198.2,Z 929.808,A -85,B 0,C 180,E1 -23902.929,E2 -23902.929} C_VEL
LIN {X 0,Y 188.849,Z 932.194,A -85,B 0,C 180,E1 -23906.067,E2 -23906.067} C_VEL
LIN {X 0,Y 184.432,Z 932.878,A -85,B 0,C 180,E1 -23907.759,E2 -23907.759} C_VEL
LIN {X 0,Y 175.233,Z 933.061,A -85,B 0,C 180,E1 -23911.951,E2 -23911.951} C_VEL
LIN {X 0,Y 169.037,Z 931.938,A -85,B 0,C 180,E1 -23915.432,E2 -23915.432} C_VEL
LIN {X 0,Y 165.757,Z 930.791,A -85,B 0,C 180,E1 -23917.567,E2 -23917.567} C_VEL
LIN {X 0,Y 160.125,Z 927.353,A -85,B 0,C 180,E1 -23922.107,E2 -23922.107} C_VEL
LIN {X 0,Y 156.775,Z 923.777,A -85,B 0,C 180,E1 -23925.726,E2 -23925.726} C_VEL
LIN {X 0,Y 154.205,Z 919.264,A -85,B 0,C 180,E1 -23929.496,E2 -23929.496} C_VEL
LIN {X 0,Y 151.959,Z 912.681,A -85,B 0,C 180,E1 -23934.027,E2 -23934.027} C_VEL
LIN {X 0,Y 150.728,Z 905.796,A -85,B 0,C 180,E1 -23937.996,E2 -23937.996} C_VEL
LIN {X 0,Y 150.198,Z 899.044,A -85,B 0,C 180,E1 -23941.341,E2 -23941.341} C_VEL
LIN {X 0,Y 150.17,Z 891.223,A -85,B 0,C 180,E1 -23944.698,E2 -23944.698} C_VEL
LIN {X 0,Y 150.735,Z 880.987,A -85,B 0,C 180,E1 -23948.378,E2 -23948.378} C_VEL
LIN {X 0,Y 151.237,Z 871.777,A -85,B 0,C 180,E1 -23951.157,E2 -23951.157} C_VEL
LIN {X 0,Y 151.915,Z 862.079,A -85,B 0,C 180,E1 -23953.65,E2 -23953.65} C_VEL
LIN {X 0,Y 152.596,Z 852.871,A -85,B 0,C 180,E1 -23955.665,E2 -23955.665} C_VEL
LIN {X 0,Y 153.206,Z 843.801,A -85,B 0,C 180,E1 -23957.348,E2 -23957.348} C_VEL
LIN {X 0,Y 153.954,Z 833.113,A -85,B 0,C 180,E1 -23958.981,E2 -23958.981} C_VEL
LIN {X 0,Y 154.578,Z 821.691,A -85,B 0,C 180,E1 -23960.371,E2 -23960.371} C_VEL
LIN {X 0,Y 155.307,Z 803.894,A -85,B 0,C 180,E1 -23962.009,E2 -23962.009} C_VEL
LIN {X 0,Y 156.896,Z 759.021,A -85,B 0,C 180,E1 -23965.778,E2 -23965.778} C_VEL
LIN {X 0,Y 151.891,Z 740.299,A -85,B 0,C 180,E1 -23967.562,E2 -23967.562} C_VEL
LIN {X 0,Y 155.208,Z 740.576,A -85,B 0,C 180,E1 -23969.944,E2 -23969.944} C_VEL
LIN {X 0,Y 157.107,Z 743.379,A -85,B 0,C 180,E1 -23971.423,E2 -23971.423} C_VEL
LIN {X 0,Y 159.048,Z 745.22,A -85,B 0,C 180,E1 -23972.75,E2 -23972.75} C_VEL
LIN {X 0,Y 161.44,Z 748.645,A -85,B 0,C 180,E1 -23974.37,E2 -23974.37} C_VEL
LIN {X 0,Y 162.772,Z 750.215,A -85,B 0,C 180,E1 -23975.197,E2 -23975.197} C_VEL
LIN {X 0,Y 166.542,Z 755.497,A -85,B 0,C 180,E1 -23977.441,E2 -23977.441} C_VEL
LIN {X 0,Y 171.747,Z 763.029,A -85,B 0,C 180,E1 -23980.224,E2 -23980.224} C_VEL
LIN {X 0,Y 177.852,Z 772.846,A -85,B 0,C 180,E1 -23983.159,E2 -23983.159} C_VEL
LIN {X 0,Y 183.449,Z 783.125,A -85,B 0,C 180,E1 -23985.621,E2 -23985.621} C_VEL
LIN {X 0,Y 186.273,Z 788.974,A -85,B 0,C 180,E1 -23986.805,E2 -23986.805} C_VEL
LIN {X 0,Y 184.907,Z 821.616,A -85,B 0,C 180,E1 -23988.208,E2 -23988.208} C_VEL
LIN {X 0,Y 183.611,Z 834.979,A -85,B 0,C 180,E1 -23989.195,E2 -23989.195} C_VEL
LIN {X 0,Y 181.531,Z 847.402,A -85,B 0,C 180,E1 -23990.481,E2 -23990.481} C_VEL
LIN {X 0,Y 178.937,Z 858.765,A -85,B 0,C 180,E1 -23992.08,E2 -23992.08} C_VEL
LIN {X 0,Y 175.595,Z 870.19,A -85,B 0,C 180,E1 -23994.156,E2 -23994.156} C_VEL
LIN {X 0,Y 172.174,Z 880.273,A -85,B 0,C 180,E1 -23996.544,E2 -23996.544} C_VEL
LIN {X 0,Y 168.673,Z 889.295,A -85,B 0,C 180,E1 -23999.293,E2 -23999.293} C_VEL
LIN {X 0,Y 164.673,Z 898.07,A -85,B 0,C 180,E1 -24002.675,E2 -24002.675} C_VEL
LIN {X 0,Y 160.87,Z 905.729,A -85,B 0,C 180,E1 -24006.555,E2 -24006.555} C_VEL
LIN {X 0,Y 157.975,Z 911.487,A -85,B 0,C 180,E1 -24010.492,E2 -24010.492} C_VEL
LIN {X 0,Y 156.393,Z 914.42,A -85,B 0,C 180,E1 -24013,E2 -24013} C_VEL
LIN {X 0,Y 154.087,Z 917.974,A -85,B 0,C 180,E1 -24016.801,E2 -24016.801} C_VEL
LIN {X 0,Y 152.98,Z 919.795,A -85,B 0,C 180,E1 -24019.394,E2 -24019.394} C_VEL
LIN {X 0,Y 151.801,Z 922.096,A -85,B 0,C 180,E1 -24024.67,E2 -24024.67} C_VEL
LIN {X 0,Y 151.251,Z 922.93,A -85,B 0,C 180,E1 -24029.982,E2 -24029.982} C_VEL
LIN {X 0,Y 151.791,Z 922.159,A -85,B 0,C 180,E1 -24035.295,E2 -24035.295} C_VEL
LIN {X 0,Y 152.949,Z 919.924,A -85,B 0,C 180,E1 -24040.573,E2 -24040.573} C_VEL
LIN {X 0,Y 154.746,Z 917.098,A -85,B 0,C 180,E1 -24044.446,E2 -24044.446} C_VEL
LIN {X 0,Y 157.079,Z 913.265,A -85,B 0,C 180,E1 -24048.233,E2 -24048.233} C_VEL
LIN {X 0,Y 159.948,Z 907.783,A -85,B 0,C 180,E1 -24052.333,E2 -24052.333} C_VEL
LIN {X 0,Y 163.416,Z 900.961,A -85,B 0,C 180,E1 -24056.136,E2 -24056.136} C_VEL
LIN {X 0,Y 167.237,Z 892.923,A -85,B 0,C 180,E1 -24059.569,E2 -24059.569} C_VEL
LIN {X 0,Y 170.67,Z 884.691,A -85,B 0,C 180,E1 -24062.345,E2 -24062.345} C_VEL
LIN {X 0,Y 174.359,Z 874.5,A -85,B 0,C 180,E1 -24065.035,E2 -24065.035} C_VEL
LIN {X 0,Y 177.707,Z 864.013,A -85,B 0,C 180,E1 -24067.163,E2 -24067.163} C_VEL
LIN {X 0,Y 180.76,Z 852.182,A -85,B 0,C 180,E1 -24069.025,E2 -24069.025} C_VEL
LIN {X 0,Y 183.179,Z 839.58,A -85,B 0,C 180,E1 -24070.489,E2 -24070.489} C_VEL
LIN {X 0,Y 184.677,Z 826.666,A -85,B 0,C 180,E1 -24071.614,E2 -24071.614} C_VEL
LIN {X 0,Y 185.498,Z 813.473,A -85,B 0,C 180,E1 -24072.331,E2 -24072.331} C_VEL
LIN {X 0,Y 186.459,Z 789.292,A -85,B 0,C 180,E1 -24073.314,E2 -24073.314} C_VEL
LIN {X 0,Y 180.246,Z 776.948,A -85,B 0,C 180,E1 -24075.975,E2 -24075.975} C_VEL
LIN {X 0,Y 173.518,Z 765.479,A -85,B 0,C 180,E1 -24079.13,E2 -24079.13} C_VEL
LIN {X 0,Y 168.04,Z 757.468,A -85,B 0,C 180,E1 -24081.973,E2 -24081.973} C_VEL
LIN {X 0,Y 165.053,Z 753.344,A -85,B 0,C 180,E1 -24083.672,E2 -24083.672} C_VEL
LIN {X 0,Y 162.264,Z 749.443,A -85,B 0,C 180,E1 -24085.389,E2 -24085.389} C_VEL
LIN {X 0,Y 159.652,Z 746.31,A -85,B 0,C 180,E1 -24087.086,E2 -24087.086} C_VEL
LIN {X 0,Y 158.559,Z 744.651,A -85,B 0,C 180,E1 -24087.867,E2 -24087.867} C_VEL
LIN {X 0,Y 156.104,Z 742.214,A -85,B 0,C 180,E1 -24089.614,E2 -24089.614} C_VEL
LIN {X 0,Y 154.742,Z 739.567,A -85,B 0,C 180,E1 -24090.775,E2 -24090.775} C_VEL
LIN {X 0,Y 152.061,Z 737.76,A -85,B 0,C 180,E1 -24092.906,E2 -24092.906} C_VEL
LIN {X 0,Y 150.505,Z 735.195,A -85,B 0,C 180,E1 -24094.428,E2 -24094.428} C_VEL
LIN {X 0,Y 150.181,Z 733.767,A -85,B 0,C 180,E1 -24094.96,E2 -24094.96} C_VEL
LIN {X 0,Y 150.304,Z 733.75,A -85,B 0,C 180,E1 -24100.894,E2 -24100.894} C_VEL
LIN {X 0,Y 150.382,Z 733.754,A -85,B 0,C 180,E1 -24106.486,E2 -24106.486} C_VEL
LIN {X 0,Y 150.589,Z 733.707,A -85,B 0,C 180,E1 -24109.241,E2 -24109.241} C_VEL
LIN {X 0,Y 150.674,Z 733.716,A -85,B 0,C 180,E1 -24111.956,E2 -24111.956} C_VEL
LIN {X 0,Y 150.873,Z 733.679,A -85,B 0,C 180,E1 -24117.33,E2 -24117.33} C_VEL
LIN {X 0,Y 151.165,Z 733.66,A -85,B 0,C 180,E1 -24120,E2 -24120} C_VEL
LIN {X 0,Y 150.614,Z 733.726,A -85,B 0,C 180,E1 -24125.355,E2 -24125.355} C_VEL
LIN {X 0,Y 150.659,Z 733.705,A -85,B 0,C 180,E1 -24128.045,E2 -24128.045} C_VEL
LIN {X 0,Y 150.55,Z 733.729,A -85,B 0,C 180,E1 -24131.493,E2 -24131.493} C_VEL
LIN {X 0,Y 150.342,Z 733.898,A -85,B 0,C 180,E1 -24138.041,E2 -24138.041} C_VEL
LIN {X 0,Y 152.342,Z 739.677,A -85,B 0,C 180,E1 -24144.532,E2 -24144.532} C_VEL
LIN {X 0,Y 153.002,Z 741.664,A -85,B 0,C 180,E1 -24146.239,E2 -24146.239} C_VEL
LIN {X 0,Y 157.774,Z 748.979,A -85,B 0,C 180,E1 -24150.075,E2 -24150.075} C_VEL
LIN {X 0,Y 162.01,Z 756.024,A -85,B 0,C 180,E1 -24153.03,E2 -24153.03} C_VEL
LIN {X 0,Y 166.634,Z 764.373,A -85,B 0,C 180,E1 -24155.91,E2 -24155.91} C_VEL
LIN {X 0,Y 169.914,Z 770.815,A -85,B 0,C 180,E1 -24157.787,E2 -24157.787} C_VEL
LIN {X 0,Y 172.648,Z 776.479,A -85,B 0,C 180,E1 -24159.262,E2 -24159.262} C_VEL
LIN {X 0,Y 177.055,Z 786.486,A -85,B 0,C 180,E1 -24161.511,E2 -24161.511} C_VEL
LIN {X 0,Y 180.731,Z 796.216,A -85,B 0,C 180,E1 -24163.313,E2 -24163.313} C_VEL
LIN {X 0,Y 182.16,Z 820.795,A -85,B 0,C 180,E1 -24165.104,E2 -24165.104} C_VEL
LIN {X 0,Y 183.108,Z 845.276,A -85,B 0,C 180,E1 -24166.675,E2 -24166.675} C_VEL
LIN {X 0,Y 181.89,Z 862.284,A -85,B 0,C 180,E1 -24167.367,E2 -24167.367} C_VEL
LIN {X 0,Y 180.06,Z 874.866,A -85,B 0,C 180,E1 -24168.183,E2 -24168.183} C_VEL
LIN {X 0,Y 177.354,Z 887.443,A -85,B 0,C 180,E1 -24169.379,E2 -24169.379} C_VEL
LIN {X 0,Y 174.132,Z 899.168,A -85,B 0,C 180,E1 -24170.927,E2 -24170.927} C_VEL
LIN {X 0,Y 170.263,Z 910.495,A -85,B 0,C 180,E1 -24172.889,E2 -24172.889} C_VEL
LIN {X 0,Y 166.196,Z 920.725,A -85,B 0,C 180,E1 -24175.211,E2 -24175.211} C_VEL
LIN {X 0,Y 162.212,Z 929.996,A -85,B 0,C 180,E1 -24177.966,E2 -24177.966} C_VEL
LIN {X 0,Y 157.993,Z 939.068,A -85,B 0,C 180,E1 -24181.454,E2 -24181.454} C_VEL
LIN {X 0,Y 154.799,Z 946.067,A -85,B 0,C 180,E1 -24184.969,E2 -24184.969} C_VEL
LIN {X 0,Y 152.816,Z 949.08,A -85,B 0,C 180,E1 -24186.727,E2 -24186.727} C_VEL
LIN {X 0,Y 148.116,Z 953.261,A -85,B 0,C 180,E1 -24189.647,E2 -24189.647} C_VEL
LIN {X 0,Y 143.837,Z 956.777,A -85,B 0,C 180,E1 -24192.876,E2 -24192.876} C_VEL
LIN {X 0,Y 142.563,Z 958.65,A -85,B 0,C 180,E1 -24195.055,E2 -24195.055} C_VEL
LIN {X 0,Y 142.079,Z 961.219,A -85,B 0,C 180,E1 -24198.608,E2 -24198.608} C_VEL
LIN {X 0,Y 142.077,Z 962.833,A -85,B 0,C 180,E1 -24201.62,E2 -24201.62} C_VEL
LIN {X 0,Y 142.357,Z 963.92,A -85,B 0,C 180,E1 -24204.353,E2 -24204.353} C_VEL
LIN {X 0,Y 142.751,Z 964.647,A -85,B 0,C 180,E1 -24207.197,E2 -24207.197} C_VEL
LIN {X 0,Y 143.207,Z 964.941,A -85,B 0,C 180,E1 -24210.019,E2 -24210.019} C_VEL
LIN {X 0,Y 142.735,Z 964.623,A -85,B 0,C 180,E1 -24212.841,E2 -24212.841} C_VEL
LIN {X 0,Y 142.349,Z 963.881,A -85,B 0,C 180,E1 -24215.685,E2 -24215.685} C_VEL
LIN {X 0,Y 142.139,Z 962.729,A -85,B 0,C 180,E1 -24218.549,E2 -24218.549} C_VEL
LIN {X 0,Y 142.429,Z 960.197,A -85,B 0,C 180,E1 -24222.848,E2 -24222.848} C_VEL
LIN {X 0,Y 143.668,Z 956.711,A -85,B 0,C 180,E1 -24227.086,E2 -24227.086} C_VEL
LIN {X 0,Y 146.396,Z 951.419,A -85,B 0,C 180,E1 -24231.86,E2 -24231.86} C_VEL
LIN {X 0,Y 148.417,Z 951.614,A -85,B 0,C 180,E1 -24235.243,E2 -24235.243} C_VEL
LIN {X 0,Y 153.243,Z 951.091,A -85,B 0,C 180,E1 -24240.315,E2 -24240.315} C_VEL
LIN {X 0,Y 159.619,Z 949.509,A -85,B 0,C 180,E1 -24244.934,E2 -24244.934} C_VEL
LIN {X 0,Y 167.387,Z 946.883,A -85,B 0,C 180,E1 -24249.052,E2 -24249.052} C_VEL
LIN {X 0,Y 176.563,Z 943.201,A -85,B 0,C 180,E1 -24252.601,E2 -24252.601} C_VEL
LIN {X 0,Y 186.741,Z 938.356,A -85,B 0,C 180,E1 -24255.665,E2 -24255.665} C_VEL
LIN {X 0,Y 197.875,Z 932.218,A -85,B 0,C 180,E1 -24258.249,E2 -24258.249} C_VEL
LIN {X 0,Y 201.526,Z 930.017,A -85,B 0,C 180,E1 -24258.959,E2 -24258.959} C_VEL
LIN {X 0,Y 201.035,Z 929.96,A -85,B 0,C 180,E1 -24259.482,E2 -24259.482} C_VEL
LIN {X 0,Y 192.924,Z 932.481,A -85,B 0,C 180,E1 -24261.736,E2 -24261.736} C_VEL
LIN {X 0,Y 188.038,Z 933.663,A -85,B 0,C 180,E1 -24263.273,E2 -24263.273} C_VEL
LIN {X 0,Y 178.661,Z 934.78,A -85,B 0,C 180,E1 -24266.584,E2 -24266.584} C_VEL
LIN {X 0,Y 170.177,Z 934.561,A -85,B 0,C 180,E1 -24270.292,E2 -24270.292} C_VEL
LIN {X 0,Y 162.663,Z 932.835,A -85,B 0,C 180,E1 -24274.402,E2 -24274.402} C_VEL
LIN {X 0,Y 156.202,Z 929.641,A -85,B 0,C 180,E1 -24278.903,E2 -24278.903} C_VEL
LIN {X 0,Y 150.935,Z 924.979,A -85,B 0,C 180,E1 -24283.777,E2 -24283.777} C_VEL
LIN {X 0,Y 148.053,Z 920.429,A -85,B 0,C 180,E1 -24287.666,E2 -24287.666} C_VEL
LIN {X 0,Y 145.545,Z 913.806,A -85,B 0,C 180,E1 -24292.369,E2 -24292.369} C_VEL
LIN {X 0,Y 144.056,Z 906.907,A -85,B 0,C 180,E1 -24296.504,E2 -24296.504} C_VEL
LIN {X 0,Y 143.356,Z 900.214,A -85,B 0,C 180,E1 -24300,E2 -24300} C_VEL
LIN {X 0,Y 143.163,Z 892.35,A -85,B 0,C 180,E1 -24303.518,E2 -24303.518} C_VEL
LIN {X 0,Y 143.627,Z 882.22,A -85,B 0,C 180,E1 -24307.38,E2 -24307.38} C_VEL
LIN {X 0,Y 144.038,Z 873.526,A -85,B 0,C 180,E1 -24310.188,E2 -24310.188} C_VEL
LIN {X 0,Y 144.655,Z 864.783,A -85,B 0,C 180,E1 -24312.598,E2 -24312.598} C_VEL
LIN {X 0,Y 145.522,Z 853.257,A -85,B 0,C 180,E1 -24315.261,E2 -24315.261} C_VEL
LIN {X 0,Y 146.297,Z 841.539,A -85,B 0,C 180,E1 -24317.473,E2 -24317.473} C_VEL
LIN {X 0,Y 147.148,Z 827.821,A -85,B 0,C 180,E1 -24319.532,E2 -24319.532} C_VEL
LIN {X 0,Y 147.973,Z 810.966,A -85,B 0,C 180,E1 -24321.324,E2 -24321.324} C_VEL
LIN {X 0,Y 149.67,Z 759.532,A -85,B 0,C 180,E1 -24325.886,E2 -24325.886} C_VEL
LIN {X 0,Y 148.34,Z 754.989,A -85,B 0,C 180,E1 -24326.349,E2 -24326.349} C_VEL
LIN {X 0,Y 148.983,Z 756.113,A -85,B 0,C 180,E1 -24326.989,E2 -24326.989} C_VEL
LIN {X 0,Y 150.04,Z 756.005,A -85,B 0,C 180,E1 -24327.794,E2 -24327.794} C_VEL
LIN {X 0,Y 151.339,Z 754.124,A -85,B 0,C 180,E1 -24328.565,E2 -24328.565} C_VEL
LIN {X 0,Y 152.977,Z 749.9,A -85,B 0,C 180,E1 -24329.311,E2 -24329.311} C_VEL
LIN {X 0,Y 153.422,Z 748.364,A -85,B 0,C 180,E1 -24329.471,E2 -24329.471} C_VEL
LIN {X 0,Y 153.914,Z 748.534,A -85,B 0,C 180,E1 -24329.824,E2 -24329.824} C_VEL
LIN {X 0,Y 156.618,Z 751.577,A -85,B 0,C 180,E1 -24331.843,E2 -24331.843} C_VEL
LIN {X 0,Y 159.516,Z 755.419,A -85,B 0,C 180,E1 -24333.86,E2 -24333.86} C_VEL
LIN {X 0,Y 165.572,Z 764.114,A -85,B 0,C 180,E1 -24337.602,E2 -24337.602} C_VEL
LIN {X 0,Y 171.351,Z 773.253,A -85,B 0,C 180,E1 -24340.723,E2 -24340.723} C_VEL
LIN {X 0,Y 176.624,Z 782.478,A -85,B 0,C 180,E1 -24343.29,E2 -24343.29} C_VEL
LIN {X 0,Y 181.126,Z 791.663,A -85,B 0,C 180,E1 -24345.348,E2 -24345.348} C_VEL
LIN {X 0,Y 179.749,Z 822.24,A -85,B 0,C 180,E1 -24346.688,E2 -24346.688} C_VEL
LIN {X 0,Y 178.397,Z 835.634,A -85,B 0,C 180,E1 -24347.688,E2 -24347.688} C_VEL
LIN {X 0,Y 176.166,Z 848.412,A -85,B 0,C 180,E1 -24349.026,E2 -24349.026} C_VEL
LIN {X 0,Y 173.447,Z 859.773,A -85,B 0,C 180,E1 -24350.654,E2 -24350.654} C_VEL
LIN {X 0,Y 169.948,Z 871.197,A -85,B 0,C 180,E1 -24352.769,E2 -24352.769} C_VEL
LIN {X 0,Y 166.356,Z 881.279,A -85,B 0,C 180,E1 -24355.21,E2 -24355.21} C_VEL
LIN {X 0,Y 162.67,Z 890.301,A -85,B 0,C 180,E1 -24358.028,E2 -24358.028} C_VEL
LIN {X 0,Y 158.463,Z 899.075,A -85,B 0,C 180,E1 -24361.508,E2 -24361.508} C_VEL
LIN {X 0,Y 154.447,Z 906.734,A -85,B 0,C 180,E1 -24365.518,E2 -24365.518} C_VEL
LIN {X 0,Y 151.369,Z 912.491,A -85,B 0,C 180,E1 -24369.604,E2 -24369.604} C_VEL
LIN {X 0,Y 149.686,Z 915.424,A -85,B 0,C 180,E1 -24372.213,E2 -24372.213} C_VEL
LIN {X 0,Y 147.253,Z 918.977,A -85,B 0,C 180,E1 -24376.176,E2 -24376.176} C_VEL
LIN {X 0,Y 146.077,Z 920.798,A -85,B 0,C 180,E1 -24378.887,E2 -24378.887} C_VEL
LIN {X 0,Y 144.805,Z 923.099,A -85,B 0,C 180,E1 -24384.411,E2 -24384.411} C_VEL
LIN {X 0,Y 144.223,Z 923.933,A -85,B 0,C 180,E1 -24389.981,E2 -24389.981} C_VEL
LIN {X 0,Y 144.795,Z 923.161,A -85,B 0,C 180,E1 -24395.552,E2 -24395.552} C_VEL
LIN {X 0,Y 146.045,Z 920.926,A -85,B 0,C 180,E1 -24401.079,E2 -24401.079} C_VEL
LIN {X 0,Y 147.951,Z 918.1,A -85,B 0,C 180,E1 -24405.125,E2 -24405.125} C_VEL
LIN {X 0,Y 150.42,Z 914.267,A -85,B 0,C 180,E1 -24409.07,E2 -24409.07} C_VEL
LIN {X 0,Y 153.47,Z 908.784,A -85,B 0,C 180,E1 -24413.33,E2 -24413.33} C_VEL
LIN {X 0,Y 157.137,Z 901.962,A -85,B 0,C 180,E1 -24417.265,E2 -24417.265} C_VEL
LIN {X 0,Y 161.161,Z 893.923,A -85,B 0,C 180,E1 -24420.802,E2 -24420.802} C_VEL
LIN {X 0,Y 164.775,Z 885.69,A -85,B 0,C 180,E1 -24423.652,E2 -24423.652} C_VEL
LIN {X 0,Y 168.652,Z 875.499,A -85,B 0,C 180,E1 -24426.406,E2 -24426.406} C_VEL
LIN {X 0,Y 172.151,Z 865.012,A -85,B 0,C 180,E1 -24428.578,E2 -24428.578} C_VEL
LIN {X 0,Y 175.358,Z 853.178,A -85,B 0,C 180,E1 -24430.47,E2 -24430.47} C_VEL
LIN {X 0,Y 177.891,Z 840.574,A -85,B 0,C 180,E1 -24431.959,E2 -24431.959} C_VEL
LIN {X 0,Y 179.48,Z 827.68,A -85,B 0,C 180,E1 -24433.103,E2 -24433.103} C_VEL
LIN {X 0,Y 180.329,Z 814.695,A -85,B 0,C 180,E1 -24433.832,E2 -24433.832} C_VEL
LIN {X 0,Y 181.298,Z 791.875,A -85,B 0,C 180,E1 -24434.784,E2 -24434.784} C_VEL
LIN {X 0,Y 175.84,Z 780.924,A -85,B 0,C 180,E1 -24437.296,E2 -24437.296} C_VEL
LIN {X 0,Y 169.907,Z 770.616,A -85,B 0,C 180,E1 -24440.269,E2 -24440.269} C_VEL
LIN {X 0,Y 164.87,Z 763.026,A -85,B 0,C 180,E1 -24443.052,E2 -24443.052} C_VEL
LIN {X 0,Y 161.78,Z 758.671,A -85,B 0,C 180,E1 -24444.925,E2 -24444.925} C_VEL
LIN {X 0,Y 159.215,Z 755.106,A -85,B 0,C 180,E1 -24446.606,E2 -24446.606} C_VEL
LIN {X 0,Y 156.519,Z 751.382,A -85,B 0,C 180,E1 -24448.524,E2 -24448.524} C_VEL
LIN {X 0,Y 153.572,Z 748.054,A -85,B 0,C 180,E1 -24450.765,E2 -24450.765} C_VEL
LIN {X 0,Y 152.409,Z 746.038,A -85,B 0,C 180,E1 -24451.793,E2 -24451.793} C_VEL
LIN {X 0,Y 149.752,Z 743.769,A -85,B 0,C 180,E1 -24454.092,E2 -24454.092} C_VEL
LIN {X 0,Y 148.121,Z 740.794,A -85,B 0,C 180,E1 -24455.843,E2 -24455.843} C_VEL
LIN {X 0,Y 144.937,Z 738.423,A -85,B 0,C 180,E1 -24459.324,E2 -24459.324} C_VEL
LIN {X 0,Y 143.583,Z 736.1,A -85,B 0,C 180,E1 -24461.263,E2 -24461.263} C_VEL
